# B&R Automation Studio project VisionSample (part 5)

#### Main.st
```iecst
// --------------------------------------------------------------------------------------------------------------------
// General vision task. This is a support task for the mappVision. The following functions are implemneted
// - Translate some values in text messages
// - Reset camera trigger when inspection is finsihed
// - Load vision application
// - Save diagnostic data
// Version 2.x (Check revision history for details)
// --------------------------------------------------------------------------------------------------------------------
PROGRAM _INIT

	userInitCommonPreAction;

	FOR idx:= START_IDX TO MAX_NUM_CAMS BY 1 DO
		setupPointersAction;

		//  Create IO path to cam
		this.path := 'IF3.ST';
		tmpStr := USINT_TO_STRING(idx);
		brsstrcat(ADR(this.path),ADR(tmpStr));

		this.recipePVName := '::Vision1:hmiInstance[';
		brsstrcat(ADR(this.recipePVName),ADR(tmpStr));
		brsstrcat(ADR(this.recipePVName),ADR('].in.recipe'));

		// Create IO path to lights
		FOR i := START_IDX TO MAX_NUM_LIGHTS BY 1 DO
			this.lightPath[i] := 'IF3.ST';
			tmpStr := USINT_TO_STRING(idx*16+(i-1));
			brsstrcat(ADR(this.lightPath[i]),ADR(tmpStr));
		END_FOR

		FOR i:= START_IDX TO MAX_NUM_RESULTS BY 1 DO
			hmi.out.tableVF.tableNum[i] := i;
		END_FOR

		hmi.out.wsPort := 18000+idx*10;
		this.mappView.enable := TRUE;
		this.mappView.wsPort := hmi.out.wsPort;
		this.mappView.simulateConfig.activate := DiagCpuIsSimulated();
		this.mappView.simulateConfig.pFile := ADR('img');
		this.mappView.simulateConfig.useRandomNumbers := FALSE;
		this.mappView.simulateConfig.appendNumber := TRUE;
		this.mappView.simulateConfig.autoIncrementNumber := TRUE;
		this.mappView.simulateConfig.minNumber := 1;
		this.mappView.simulateConfig.maxNumber := 3;

		this.visionDiagFileDevice := 'VI_DIAG'; // File device is created in Files program (changes to USB if such is pluged in)

		hmi.out.camera.plNodeNr := idx;
		hmi.in.recipe.cam.focus := 200;
		hmi.in.recipe.cam.exposureTime := 100;

		hmi.in.cmd.resetInfo := TRUE;

		// -----------------------------------------------------------------------------------------------------------
		// Set camera specific data
		// -----------------------------------------------------------------------------------------------------------

		hmi.in.cmd.resultTabIndex := 5;
		CASE idx OF
			1:
				this.mappView.pMappLink := ADR(gCameraBlob);
				this.mappView.simulateConfig.pDevice := ADR('SIM_BLOB');
				hmi.out.camera.visionFunction := 'BLOB';
				hmi.out.usedVF.BLOB := TRUE;
				hmi.in.cmd.resultTabIndex := MIN(hmi.in.cmd.resultTabIndex,idx-1);
			2:
				this.mappView.pMappLink := ADR(gCameraCodeReading);
				this.mappView.simulateConfig.pDevice := ADR('SIM_CR');
				hmi.out.camera.visionFunction := 'Code Reader';
				hmi.out.usedVF.codeReader := TRUE;
				hmi.in.cmd.resultTabIndex := MIN(hmi.in.cmd.resultTabIndex,idx-1);
				(*hmi.out.VF.numResults*)
			3:
				this.mappView.pMappLink := ADR(gCameraMatch);
				this.mappView.simulateConfig.pDevice := ADR('SIM_MATCH');
				hmi.out.camera.visionFunction := 'Matching';
				hmi.out.usedVF.matching := TRUE;
				hmi.in.cmd.resultTabIndex := MIN(hmi.in.cmd.resultTabIndex,idx-1);
			4:
				this.mappView.pMappLink := ADR(gCameraMeasurement);
				this.mappView.simulateConfig.pDevice := ADR('SIM_MEAS');
				hmi.out.camera.visionFunction := 'Measurement';
				hmi.out.usedVF.measurement := TRUE;
				hmi.in.cmd.resultTabIndex := MIN(hmi.in.cmd.resultTabIndex,idx-1);
			5:
				this.mappView.pMappLink := ADR(gCameraOCR);
				this.mappView.simulateConfig.pDevice := ADR('SIM_OCR');
				hmi.out.camera.visionFunction := 'OCR';
				hmi.out.usedVF.OCR := TRUE;
				hmi.in.cmd.resultTabIndex := MIN(hmi.in.cmd.resultTabIndex,idx-1);
			6:
				this.mappView.pMappLink := ADR(gCameraPxl);
				this.mappView.simulateConfig.pDevice := ADR('SIM_PXCNT');
				hmi.out.camera.visionFunction := 'Pixel Counter';
				hmi.out.usedVF.pixelCounter := TRUE;
				hmi.in.cmd.resultTabIndex := MIN(hmi.in.cmd.resultTabIndex,idx-1);

		END_CASE

		userInitLocalPostAction;

	END_FOR

END_PROGRAM

// -----------------------------------------------------------------------------------------------------------
// Cyclic part
// -----------------------------------------------------------------------------------------------------------
PROGRAM _CYCLIC

	userCommonPreAction; // user common action before all other

	FOR idx:= START_IDX TO MAX_NUM_CAMS BY 1 DO
		setupPointersAction;

		userLocalPreAction; // user local action before all other

		// -----------------------------------------------------------------------------------------------------------
		// Translate camera status in readable text
		// -----------------------------------------------------------------------------------------------------------
		IF hw.camera.in.common.moduleOk THEN
			brdkViBase_camStatusToString(hw.camera.in.status.cameraStatus,ADR(hmi.out.camera.statusText));
		ELSE
			hmi.out.camera.statusText := 'Disconnected';
		END_IF

		// -----------------------------------------------------------------------------------------------------------
		// Check if vision cockpit is open
		// -----------------------------------------------------------------------------------------------------------
		hmi.out.camera.mappVisionActive := (hw.camera.in.status.cameraStatus AND 16#8000_0000) > 0;

		// -----------------------------------------------------------------------------------------------------------
		// Read camera hardware info
		// -----------------------------------------------------------------------------------------------------------

		IF hmi.in.cmd.resetInfo THEN
			hmi.in.cmd.resetInfo := FALSE;
			hmi.in.cameraInfo.distance := hmi.in.recipe.cam.focus;
			this.brdkViBase_getCameraInfo_0.execute := TRUE;
			this.brdkViBase_getCameraInfo_0.pluggedModule := hw.camera.in.common.moduleOk AND NOT DiagCpuIsSimulated();

			FOR i := START_IDX TO MAX_NUM_LIGHTS BY 1 DO
				this.brdkViBase_getLightInfo[i].execute := TRUE;
				this.brdkViBase_getLightInfo[i].pInfo := ADR(hmi.out.lights[i].info);
				this.brdkViBase_getLightInfo[i].pDevicePath := ADR(this.lightPath[i]);
				this.brdkViBase_getLightInfo[i].pluggedModule := hw.lights[i].in.common.moduleOk AND NOT DiagCpuIsSimulated();
			END_FOR

		END_IF

		this.brdkViBase_getCameraInfo_0.pDevicePath := ADR(this.path);
		this.brdkViBase_getCameraInfo_0.pInfo := ADR(hmi.in.cameraInfo);
		this.brdkViBase_getCameraInfo_0();

		FOR i:=START_IDX TO MAX_NUM_LIGHTS BY 1 DO
			this.brdkViBase_getLightInfo[i]();

			IF hmi.out.lights[i].info.orderNr <> '' AND this.brdkViBase_getLightInfo[i].status = ERR_OK THEN
				// set Camera flash options based on current camera
				brdkViBase_LEDColorToOptions(hmi.out.lights[i].info.LED_color, ADR(hmi.out.lights[i].flashLightOptions));
			END_IF
		END_FOR

		IF hw.camera.out.par.focus <> hmi.in.recipe.cam.focus THEN
			hmi.in.cameraInfo.distance := hmi.in.recipe.cam.focus;
		END_IF

		IF hmi.in.cameraInfo.orderNr <> '' AND this.brdkViBase_getCameraInfo_0.status = ERR_OK THEN
			brdkViBase_calcOpticInfo(hmi.in.cameraInfo, hmi.out.camera.opticInfo); // calculate optic info based on defined info

			// set Camera flash options based on current camera
			brdkViBase_LEDColorToOptions(hmi.in.cameraInfo.LED_color, ADR(hmi.out.camera.flashLightOptions));
		END_IF

		IF hw.io.in.nettime > this.axisTrig.nettimeLastCycle_us THEN
			this.axisTrig.powerlinkCycle_us	:= hw.io.in.nettime - this.axisTrig.nettimeLastCycle_us;
		ELSE
			this.axisTrig.powerlinkCycle_us	:= -2147483648-hw.io.in.nettime + 2147483647-this.axisTrig.nettimeLastCycle_us; // handle wrap around
		END_IF
		this.axisTrig.nettimeLastCycle_us	:= hw.io.in.nettime;

		// -----------------------------------------------------------------------------------------------------------
		// Image trigger (camera and lights)
		// -----------------------------------------------------------------------------------------------------------
		hmi.in.recipe.cam.flashColor := STRING_TO_USINT(hmi.in.recipe.cam.flashColorStr);
		hw.camera.out.par.focus 			:= hmi.in.recipe.cam.focus;
		hw.camera.out.par.flashSegment	 	:= hmi.in.recipe.cam.flashSegment;
		hw.camera.out.par.flashColor 		:= hmi.in.recipe.cam.flashColor;
		hw.camera.out.par.exposureTime 		:= hmi.in.recipe.cam.exposureTime;
		hw.camera.out.par.chromaticLock 	:= hmi.in.recipe.cam.chromaticLock;
		hw.camera.out.par.gainLevel 		:= hmi.in.recipe.cam.gainLevel;
		hw.camera.out.par.IRFilter			:= hmi.in.recipe.cam.IRFilter;

		//-------------------------------------------------------------------------

		// Copy recipe data (e.g. enable, maximal number of results, etc.)
		hw.VF.blob.out			:=hmi.in.recipe.BLOB;
		hw.VF.codeReader.out	:= hmi.in.recipe.CR;
		hw.VF.matching.out		:=hmi.in.recipe.match;
		hw.VF.measurement.out	:=hmi.in.recipe.meassurement;
		hw.VF.ocr.out			:=hmi.in.recipe.OCR;
		hw.VF.pixelCnt.out		:=hmi.in.recipe.pxCnt;

		hmi.out.camera.processingTime:=hw.camera.in.status.cameraProcessingTime;

		CASE idx OF
			1:
				hmi.out.VF.processingTime := hw.VF.blob.in.common.functionProcessingTime;
				hmi.out.VF.numResults := hw.VF.blob.in.common.numResults;
			2:
				hmi.out.VF.processingTime := hw.VF.codeReader.in.common.functionProcessingTime;
				hmi.out.VF.numResults := hw.VF.codeReader.in.common.numResults;
			3:
				hmi.out.VF.processingTime := hw.VF.matching.in.common.functionProcessingTime;
				hmi.out.VF.numResults := hw.VF.matching.in.common.numResults;
			4:
				hmi.out.VF.processingTime := hw.VF.measurement.in.common.functionProcessingTime;
				hmi.out.VF.numResults := hw.VF.measurement.in.common.numResults;
			5:
				hmi.out.VF.processingTime := hw.VF.ocr.in.common.functionProcessingTime;
				hmi.out.VF.numResults := hw.VF.ocr.in.common.numResults;
			6:
				hmi.out.VF.processingTime := hw.VF.pixelCnt.in.common.functionProcessingTime;
				hmi.out.VF.numResults := hw.VF.pixelCnt.in.common.numResults;
		END_CASE;

		//-------------------------------------------------------------------------

		this.ioTrigger(CLK := hw.io.in.commonTrigger OR NOT hw.io.in.individualTrigger);
		this.repetitiveTriggerTON.IN := hmi.in.recipe.repetitiveTrigger;
		this.repetitiveTriggerTON.PT := UDINT_TO_TIME(hmi.in.recipe.repetitiveTriggerInterval);
		this.repetitiveTriggerTON();

		// check if camera is ready for an image trigger and MappView have been updated
		IF this.brdkViBase_imgTrigger_0.ready AND NOT this.brdkViBase_imgTrigger_0.busy AND this.mappView.status = 0 THEN

			// Hmi manual trigger
			IF hmi.in.cmd.trigger OR this.repetitiveTriggerTON.Q THEN
				hmi.in.cmd.trigger 							:= FALSE;

				this.repetitiveTriggerTON(IN:=FALSE);

				this.brdkViBase_imgTrigger_0.trigger 		:= TRUE;
				this.brdkViBase_imgTrigger_0.delayNettime 	:= hw.io.in.nettime + gAxis.status.powerlinkCycleTime * 12+10000; // Calc nettime close to currnet time
				this.currentTriggerNum := 1;
				// Axis trigger
			ELSIF hmi.in.recipe.enableAxisTrigger AND
				gAxis.status.triggerTimeDelta >= (commonHmi.in.recipe.visionPreTriggerCycles * this.axisTrig.powerlinkCycle_us) AND
				gAxis.status.triggerTimeDelta <= ((commonHmi.in.recipe.visionPreTriggerCycles + 1) * this.axisTrig.powerlinkCycle_us) THEN

				this.brdkViBase_imgTrigger_0.trigger := TRUE;
				this.brdkViBase_imgTrigger_0.delayNettime := gAxis.status.nettime + gAxis.status.triggerTimeDelta; // Use time calculated in Axis program
			ELSIF hmi.in.recipe.enableIoTrigger AND this.ioTrigger.Q THEN

				this.brdkViBase_imgTrigger_0.trigger := TRUE;
				this.brdkViBase_imgTrigger_0.delayNettime :=  hw.io.in.nettime + hmi.in.recipe.ioTriggerDelay ; // Use time calculated in Axis program

			ELSIF this.currentTriggerNum < hmi.in.recipe.multiCaptureNum AND NOT hmi.in.recipe.repetitiveTrigger THEN

				this.brdkViBase_imgTrigger_0.trigger 		:= TRUE;
				this.brdkViBase_imgTrigger_0.delayNettime 	:= hw.io.in.nettime + gAxis.status.powerlinkCycleTime * 12+10000; // Calc nettime close to currnet time

				this.currentTriggerNum := 		this.currentTriggerNum +1;

			END_IF
		END_IF

		this.brdkViBase_imgTrigger_0.searchAcquisitonSettings := hmi.in.cmd.autoSearch;
		this.brdkViBase_imgTrigger_0.pCameraHw := ADR(hw.camera);
		this.brdkViBase_imgTrigger_0.numLights := MAX_NUM_LIGHTS;
		this.brdkViBase_imgTrigger_0.pLightHw := ADR(hw.lights);
		this.brdkViBase_imgTrigger_0.useCamColorForLight := hmi.in.recipe.useCamLedColorForLight;
		this.brdkViBase_imgTrigger_0.useCamExpTimeForLight := hmi.in.recipe.useCamExpTimeForLight;
		this.brdkViBase_imgTrigger_0.simulate.enable := DiagCpuIsSimulated();
		this.brdkViBase_imgTrigger_0.simulate.alwaysSimulateNonePresentLights := TRUE;
		this.brdkViBase_imgTrigger_0.simulate.imgProcessingDelay := T#300ms;
		this.brdkViBase_imgTrigger_0();

		FOR i:=START_IDX TO MAX_NUM_LIGHTS BY 1 DO

			// Manual Light trigger
			// exposuretime
			IF hmi.in.recipe.useCamExpTimeForLight THEN
				hw.lights[i].out.par.exposureTime := hmi.in.recipe.cam.exposureTime;
			ELSE
				hw.lights[i].out.par.exposureTime := hmi.in.recipe.lights[i].exposureTime;
			END_IF
			// color
			IF hmi.in.recipe.useCamLedColorForLight THEN
				hw.lights[i].out.par.flashColor := hmi.in.recipe.cam.flashColor;
			ELSE
				hw.lights[i].out.par.flashColor := hmi.in.recipe.lights[i].flashColor;
			END_IF

			hmi.out.lights[i].common:=hw.lights[i].in.common;
			hmi.out.lights[i].status:=hw.lights[i].in.status;
			hw.lights[i].out.par.flashAngle:=hmi.in.recipe.lights[i].flashAngle;

			hmi.out.lights[i].plNodeNr := idx*16+UINT_TO_USINT(i-1);

			IF hmi.in.cmd.lights[i].flashTrigger AND NOT hw.lights[i].out.cmd.flashTrigger THEN
				hmi.in.cmd.lights[i].flashTrigger := FALSE;
				hw.lights[i].out.cmd.flashTrigger := TRUE;

				// Nettime
				hw.lights[i].out.par.nettime := hw.io.in.nettime + gAxis.status.powerlinkCycleTime * commonHmi.in.recipe.visionPreTriggerCycles;
			ELSIF 	hw.lights[i].out.cmd.flashTrigger AND hw.lights[i].out.par.nettime <= hw.io.in.nettime THEN
				hw.lights[i].out.cmd.flashTrigger := FALSE;
			END_IF
		END_FOR

		// -----------------------------------------------------------------------------------------------------------
		// New image ready and results
		// -----------------------------------------------------------------------------------------------------------
		// New image (hight for one scan)
		IF this.brdkViBase_imgTrigger_0.newImage THEN

			this.mappView.updateImage := NOT hmi.in.recipe.showOnlyLastImage OR this.currentTriggerNum = hmi.in.recipe.multiCaptureNum; // Trigger an update of the image on hmi
			this.DTGetTime_0(enable := TRUE);

			processResultsAction; // Process results action

			userResultProcessingAction; // User defined process results

		END_IF

		// -----------------------------------------------------------------------------------------------------------
		// Selection of specific result
		// -----------------------------------------------------------------------------------------------------------
		IF hmi.in.cmd.click THEN
			hmi.in.cmd.click := FALSE;

			//VF
			brdkStrSubStr(ADR(tmpVF),ADR(hmi.in.cmd.elemId),1,1);
			//ID
			brsstrcpy(ADR(tmpID),ADR(hmi.in.cmd.elemId)+2);

			hmi.in.cmd.intElemId := STRING_TO_USINT(tmpID);
			IF hmi.in.cmd.intElemId > MAX_NUM_RESULTS THEN
				hmi.in.cmd.intElemId := 0;
			END_IF

		END_IF

		IF hmi.in.cmd.intElemId <> this.oldIntElemID THEN
			this.oldIntElemID := hmi.in.cmd.intElemId;
			processResultsAction;
		END_IF

		// -----------------------------------------------------------------------------------------------------------
		// Auto search vision acquistion settings done (save found settings in recipe structure)
		// -----------------------------------------------------------------------------------------------------------

		// search Auto Focus done (hight for one scan)
		IF this.brdkViBase_imgTrigger_0.searchAcquisitonSettingsDone THEN
			hmi.in.cmd.autoSearch 			:= FALSE;
			hmi.in.recipe.cam.gainLevel 	:=	 hw.camera.in.status.gainLevel;
			hmi.in.recipe.cam.focus		 	:=	 hw.camera.in.status.focus;
			hmi.in.recipe.cam.exposureTime 	:=	 hw.camera.in.status.exposureTime;
			this.brdkViBase_imgTrigger_0.searchAcquisitonSettings := FALSE;
			hmi.in.cmd.trigger 				:= TRUE;
		END_IF

		// -----------------------------------------------------------------------------------------------------------
		// MappView get image to show om hmi
		// -----------------------------------------------------------------------------------------------------------

		IF DiagCpuIsSimulated() THEN
			this.mappView.imageFormat := BRDKVIIMG_IMG_TYPE_JPEG;
		ELSE
			this.mappView.imageFormat := commonHmi.in.recipe.imageFormat;
		END_IF
		this.mappView.jpegQuality := commonHmi.in.recipe.jpegQuality;
		this.mappView();

		// -----------------------------------------------------------------------------------------------------------
		// Save image to file devive F:/images
		// -----------------------------------------------------------------------------------------------------------
		CASE this.saveState OF
			0:

				IF (hmi.in.cmd.saveImage OR (this.mappView.newSvgReady AND commonHmi.in.recipe.saveAllImages))  AND gFiles.output.ready THEN
					hmi.in.cmd.saveImage := FALSE;

					// create filename with VF name and current date of the image
					brsstrcpy(ADR(this.tmpFileName),ADR(hmi.out.camera.visionFunction));
					brsstrcat(ADR(this.tmpFileName),ADR('-'));
					brdkViBase_dateTimeToString(this.DTGetTime_0.DT1,'%Y-%m-%d-%H-%M-%S',ADR(this.tmpFileName));

					brsstrcpy(ADR(this.brdkFileWrite.fileName),ADR(this.tmpFileName));

					CASE this.mappView.imageFormat OF
						BRDKVIIMG_IMG_TYPE_JPEG:
							brsstrcat(ADR(this.brdkFileWrite.fileName),ADR('.jpg'));
						BRDKVIIMG_IMG_TYPE_BMP:
							brsstrcat(ADR(this.brdkFileWrite.fileName),ADR('.bmp'));
					END_CASE

					this.brdkFileWrite.enable := TRUE;
					this.brdkFileWrite.dataLength := this.mappView.internal.getImage.destLen;
					this.brdkFileWrite.pData := this.mappView.internal.getImage.pDest;
					this.brdkFileWrite.overwrite := TRUE;
					this.brdkFileWrite.fileDevice := 'IMG';

					this.saveState := 10;
				END_IF
			10:

				IF this.brdkFileWrite.done THEN
					gFiles.input.refresh := TRUE;
					this.brdkFileWrite.enable := FALSE;
					this.saveState := 20;
				END_IF

			20:
				brsstrcpy(ADR(this.brdkFileWrite.fileName),ADR(this.tmpFileName));

				brsstrcat(ADR(this.brdkFileWrite.fileName),ADR('.svg'));
				this.brdkFileWrite.enable := TRUE;
				this.brdkFileWrite.dataLength := brsstrlen(ADR(hmi.out.svgOverlay));
				this.brdkFileWrite.pData := ADR(hmi.out.svgOverlay);
				this.brdkFileWrite.overwrite := TRUE;
				this.brdkFileWrite.fileDevice := 'IMG';

				this.saveState := 30;

			30:
				IF this.brdkFileWrite.done THEN
					gFiles.input.refresh := TRUE;
					this.brdkFileWrite.enable := FALSE;
					this.saveState := 0;
				END_IF

		END_CASE

		this.brdkFileWrite();

		// -----------------------------------------------------------------------------------------------------------
		// Save diagnostic data
		// -----------------------------------------------------------------------------------------------------------
		IF hmi.in.cmd.saveDiagnositc AND gFiles.output.ready THEN
			hmi.in.cmd.saveDiagnositc 			:= FALSE;

			// Delete old file first
			this.fileDelete.enable 					:= TRUE;
			this.fileDelete.pDevice 				:= ADR(this.visionDiagFileDevice);
			this.fileDelete.pName 					:= ADR(hmi.in.diagnosticFilename);

			// Upload diagnostic information
			this.viBaseSaveDiagData_0.MpLink 		:= this.mappView.pMappLink;
			this.viBaseSaveDiagData_0.DeviceName 	:= ADR(this.visionDiagFileDevice);
			this.viBaseSaveDiagData_0.FileName 		:= ADR(hmi.in.diagnosticFilename);
			hmi.out.camera.saveDiagStatus 			:= UINT_TO_DINT(ERR_FUB_BUSY);
		END_IF

		// file delete done or error (if file do not exsist)
		IF (this.fileDelete.enable AND this.fileDelete.status = ERR_OK) THEN
			this.fileDelete.enable 				:= FALSE;
			this.viBaseSaveDiagData_0.Execute 	:= TRUE;
		END_IF

		// Done
		IF (this.viBaseSaveDiagData_0.Done) THEN
			hmi.out.camera.saveDiagStatus		:= UINT_TO_DINT(ERR_OK);
			this.viBaseSaveDiagData_0.Execute 	:= FALSE;
		END_IF

		// Error
		IF (NOT this.viBaseSaveDiagData_0.Busy AND this.viBaseSaveDiagData_0.Error) THEN
			hmi.out.camera.saveDiagStatus		:= this.viBaseSaveDiagData_0.StatusID;
			this.viBaseSaveDiagData_0.Execute 	:= FALSE;
		END_IF

		this.viBaseSaveDiagData_0();
		this.fileDelete();

		// -----------------------------------------------------------------------------------------------------------
		// Get Vision application list from camera
		// -----------------------------------------------------------------------------------------------------------

		// trigger
		IF hmi.in.cmd.vaList.refresh THEN
			hmi.in.cmd.vaList.refresh 	:= FALSE;

			this.getVaList.Execute 		:= TRUE;
			this.getVaList.Format 		:= viBASE_FORMAT_PLAIN_TEXT;
			this.getVaList.List 		:= ADR(hmi.out.vaList.list);
			this.getVaList.ListLen 		:= SIZEOF(hmi.out.vaList.list);
			this.getVaList.MpLink 		:= this.mappView.pMappLink;
		END_IF

		// Done
		IF this.getVaList.Done THEN
			this.getVaList.Execute 		:= FALSE;
			hmi.out.vaList.length 		:= this.getVaList.NrEntries;
		END_IF

		// Error
		IF this.getVaList.Error THEN
			this.getVaList.Execute 		:= FALSE;
			hmi.out.vaList.lastError 	:= this.getVaList.StatusID;
		END_IF

		this.getVaList();

		// -----------------------------------------------------------------------------------------------------------
		// Load vision application
		// -----------------------------------------------------------------------------------------------------------

		// Trigger
		IF hmi.in.cmd.vaList.load AND brsstrlen(ADR(hmi.out.vaList.list[hmi.in.cmd.vaList.selectedIndex])) > 5 THEN
			hmi.in.cmd.vaList.load 						:= FALSE;

			this.viBaseLoadApplication_0.Execute 	:= TRUE;
			this.viBaseLoadApplication_0.MpLink		:= this.mappView.pMappLink;
			this.viBaseLoadApplication_0.Name		:= ADR(hmi.out.vaList.list[hmi.in.cmd.vaList.selectedIndex]);
			hmi.out.camera.vaLoad 					:= UINT_TO_DINT(ERR_FUB_BUSY);
		ELSE
			hmi.in.cmd.vaList.load := FALSE;
		END_IF

		// Done
		IF (this.viBaseLoadApplication_0.Done) THEN
			hmi.in.cmd.vaList.selectedIndex := 0;
			this.viBaseLoadApplication_0.Execute 	:= FALSE;
			hmi.out.camera.vaLoad 					:= UINT_TO_DINT(ERR_OK);
		END_IF

		// Error
		IF (NOT this.viBaseLoadApplication_0.Busy AND this.viBaseLoadApplication_0.Error) THEN
			this.viBaseLoadApplication_0.Execute 	:= FALSE;
			hmi.out.camera.vaLoad 					:= this.viBaseLoadApplication_0.StatusID;
		END_IF

		this.viBaseLoadApplication_0();

		// -----------------------------------------------------------------------------------------------------------
		// HMI stuff
		// -----------------------------------------------------------------------------------------------------------
		hmiAction;

		// -----------------------------------------------------------------------------------------------------------
		// Recipe handling (register recipse data structure
		// -----------------------------------------------------------------------------------------------------------
		this.mpRecipeRegVar.Enable 		:= gRecipe.out.active;
		this.mpRecipeRegVar.MpLink 		:= gRecipe.out.mpLink;
		this.mpRecipeRegVar.ConfirmSave := this.mpRecipeRegVar.SaveNotification;
		this.mpRecipeRegVar.Category 	:= ADR('Recipe');
		this.mpRecipeRegVar.PVName 		:= ADR(this.recipePVName);
		this.mpRecipeRegVar();

		// handle conversion from CR dropDown value to interger and back
		IF this.mpRecipeRegVar.UpdateNotification THEN
			hmi.in.recipe.CRTypeStr := USINT_TO_STRING(hmi.in.recipe.CR.symbolType);

			FOR i:=START_IDX TO MAX_NUM_LIGHTS BY 1 DO
				this.brdkViBase_getLightInfo[i]();
				hmi.in.cmd.lightColorStr[i] := USINT_TO_STRING(hmi.in.recipe.lights[i].flashColor );
			END_FOR

		ELSE
			hmi.in.recipe.CR.symbolType := STRING_TO_USINT(hmi.in.recipe.CRTypeStr);
			FOR i:=START_IDX TO MAX_NUM_LIGHTS BY 1 DO
				this.brdkViBase_getLightInfo[i]();
				hmi.in.recipe.lights[i].flashColor := STRING_TO_USINT(hmi.in.cmd.lightColorStr[i]);
			END_FOR
		END_IF

		// Clear ready for init (auto load) if data structures have not been registred
		IF NOT this.mpRecipeRegVar.Active THEN
			gRecipe.in.readyForInit := FALSE;
		END_IF

		userLocalPostAction; // user local action after all other

	END_FOR

	userCommonPostAction; // user common action after all other

	// -----------------------------------------------------------------------------------------------------------
	//Configure the pointers (this,hmi,hw etc.) show the correct data for that watch index
	// -----------------------------------------------------------------------------------------------------------
	watchIdx := LIMIT(START_IDX,watchIdx,MAX_NUM_CAMS);
	idx := watchIdx;
	setupPointersAction;

					END_PROGRAM

PROGRAM _EXIT

	FOR idx:= START_IDX TO MAX_NUM_CAMS BY 1 DO
		setupPointersAction;

		this.mappView(enable := FALSE);
		this.mpRecipeRegVar(Enable := FALSE);

		userExitLocalPostAction;
	END_FOR

	userExitCommonPostAction;

					END_PROGRAM
```

### VisionTypes.typ
```iecst
(*-----------------------------------------------------------------------------------------------------------------------------------------*)
(*General vision structures*)

TYPE
	typVisionMain : 	STRUCT
		CMD : typVisionCommand;
		CFG : typVisionConfig;
		DAT : typVisionData;
		HW : typVisionHW;
	END_STRUCT;
	typVisionCommand : 	STRUCT
		ImageTrigger : BOOL;
		ImageTriggerReset : BOOL;
		AutoSetupStartStop : BOOL;
	END_STRUCT;
	typVisionConfig : 	STRUCT
		VisionFunction : enumVisionFunction;
		PowerlinkNode : USINT;
		DataStructure : UDINT;
		ComponentLink : ViComponentType;
		ResolutionWidth : UINT; (*Nr of sensor pixels in x direction (width). Is always bigger than height*)
		ResolutionHeight : UINT; (*Nr of sensor pixels in y direction (height). Is always smaller than width*)
	END_STRUCT;
	typVisionData : 	STRUCT
		Enable : BOOL := FALSE;
		MaxItemCnt : USINT := 10;
		NettimeDelay : DINT;
		Timeout : UINT := 5000;
		Gain : USINT;
		Focus : UINT;
		Exposure : UDINT;
		FlashColor : USINT := 1;
		FlashSegment : USINT := 15;
		LedColor : USINT;
		IRFilter : BOOL;
		OffsetROIX : DINT;
		OffsetROIY : DINT;
		OffsetROIRotationCenterX : DINT;
		OffsetROIRotationCenterY : DINT;
		OffsetROIOrientation : INT;
		ChromaticLock : BOOL;
		Alignment : USINT;
		AutoSetupGain : USINT;
		AutoSetupFocus : UINT;
		AutoSetupExposure : UDINT;
		AcquisitionAcceptedCnt : USINT;
		AcquisitionCompletedCnt : USINT;
		AcquisitionFailedCnt : USINT;
		LightWarningCnt : USINT;
		ImageProcessingError : UINT;
		ImageProcessingActive : BOOL;
		ImageNettime : DINT;
		ProcessingTimeCamera : UINT;
		ProcessingTimeFunction : UINT;
		ResultCnt : USINT;
		CockpitIsActive : BOOL;
		Status : UDINT;
		StatusText : STRING[30];
		Active : BOOL;
	END_STRUCT;
	typVisionHW : 	STRUCT
		Connected : BOOL;
		Ready : BOOL;
		DigitalInput01 : BOOL;
		DigitalOutput01 : BOOL;
		DigitalOutputStatus01 : BOOL;
		DigitalOutput02 : BOOL;
		DigitalOutputStatus02 : BOOL;
		SerialNumber : UDINT;
		ID : UDINT;
		Variant : UDINT;
		Firmware : UDINT;
		Undervoltage : BOOL;
		Temperature : SINT;
	END_STRUCT;
	enumVisionFunction :
		(
		enumFunctionNone,
		enumBlob,
		enumCoderReader,
		enumMatch,
		enumMeasurement,
		enumOCR,
		enumDOCR,
		enumPixelCounter
		);
END_TYPE

(*-----------------------------------------------------------------------------------------------------------------------------------------*)
(*General Light structures*)

TYPE
	typLightMain : 	STRUCT
		CMD : typLightCommand;
		CFG : typLightConfig;
		DAT : typLightData;
		HW : typLightHW;
	END_STRUCT;
	typLightCommand : 	STRUCT
		FlashTrigger : BOOL;
		FlashTriggerReset : BOOL;
	END_STRUCT;
	typLightConfig : 	STRUCT
		LightType : enumLightType;
		PowerlinkNode : USINT;
	END_STRUCT;
	typLightData : 	STRUCT
		Enable : USINT := 1;
		FlashColor : USINT := 1;
		FlashSegment : UINT := 15;
		Exposure : UDINT := 200;
		SetAngle : UINT;
		Timeout : UINT := 5000;
		NettimeDelay : DINT;
		FlashAcceptedCnt : USINT;
		FlashCompletedCnt : USINT;
		FlashFailedCnt : USINT;
		Status : UDINT;
	END_STRUCT;
	typLightHW : 	STRUCT
		Connected : BOOL;
		Ready : BOOL;
		SerialNumber : UDINT;
		ID : UDINT;
		Variant : UDINT;
		Firmware : UDINT;
		TemperatureLED : SINT;
		TemperatureControllerBoard : SINT;
		WarningCnt : USINT;
	END_STRUCT;
	enumLightType :
		(
		enumLightNone,
		enumBacklight,
		enumLightbar
		);
END_TYPE

(*-----------------------------------------------------------------------------------------------------------------------------------------*)
(*General nettime structures*)

TYPE
	typVisionNettime : 	STRUCT
		CMD : typNettimeCommand;
		CFG : typNettimeConfig;
		DAT : typNettimeData;
	END_STRUCT;
	typNettimeCommand : 	STRUCT
		Activate : BOOL;
	END_STRUCT;
	typNettimeConfig : 	STRUCT
		AxisPeriod : LREAL; (*Units when period repeats*)
		AxisPositionTrigger : LREAL; (*Position in the period where trigger is fired*)
		AxisPositionDelay_Cycles : LREAL; (*Delay in PLK cycles for the read position from drive*)
		VisionPreTrigger_Cycles : DINT; (*Number of powerlink cycles the trigger has to be send ahead*)
	END_STRUCT;
	typNettimeData : 	STRUCT
		NettimeNext_us : DINT; (*Calculated nettime for next trigger*)
		NettimeDelta_us : DINT; (*Difference between current nettime and calculated nettime for the camera trigger*)
		AxisPosition : LREAL; (*Current axis position*)
		AxisVelocity : LREAL; (*Current axis position*)
		AxisInVelocity : BOOL; (*Indicates that the axis is moving at speed*)
		Overflow : DINT; (*Counts up when a trigger could not be set on time*)
	END_STRUCT;
END_TYPE

(*-----------------------------------------------------------------------------------------------------------------------------------------*)
(*Image upload structures*)

TYPE
	typVisionImage : 	STRUCT
		CMD : typVisionImageCommand;
		CFG : typVisionImageConfig;
		DAT : typVisionImageData;
	END_STRUCT;
	typVisionImageCommand : 	STRUCT
		CreateDir : BOOL;
		DeleteDir : BOOL;
		DeleteImage : BOOL;
		GetImage : BOOL;
		SaveImage : BOOL;
		Refresh : BOOL;
		ResetError : BOOL;
	END_STRUCT;
	typVisionImageConfig : 	STRUCT
		FileDevice : STRING[80];
		FileName : STRING[80];
		DirName : STRING[80];
		ImageQuality : USINT := 50;
		ImageHeight : UINT := 1280;
		ImageWidth : UINT := 1024;
		ImageType : ViBaseImageTypeEnum;
		ComponentLink : ViComponentType;
	END_STRUCT;
	typVisionImageData : 	STRUCT
		ImagesList : ARRAY[0..19]OF STRING[80];
		ImageSelected : STRING[80];
		ImagePath : STRING[80];
		Crosshair : ARRAY[1..MAX_NUM_RESULTS]OF typVisionImageDataCrosshair;
		Status : DINT;
	END_STRUCT;
	typVisionImageDataCrosshair : 	STRUCT
		CrosshairX : REAL;
		CrosshairY : REAL;
		CrosshairRotate : REAL;
		Text : STRING[1000];
	END_STRUCT;
END_TYPE

(*-----------------------------------------------------------------------------------------------------------------------------------------*)
(*Vision specific structures*)

TYPE
	typCodeReaderMain : 	STRUCT  (*Code reader structures*)
		CodeType : USINT;
		GradingEnable : BOOL;
		RobustnessEnable : BOOL;
		ParameterMode : USINT;
		ParameterOptimization : USINT;
		BarcodeText : ARRAY[1..MAX_NUM_RESULTS]OF STRING[100];
		BarcodeType : ARRAY[1..MAX_NUM_RESULTS]OF USINT;
		PositionX : ARRAY[1..MAX_NUM_RESULTS]OF DINT;
		PositionY : ARRAY[1..MAX_NUM_RESULTS]OF DINT;
		Orientation : ARRAY[1..MAX_NUM_RESULTS]OF INT;
		Grading : ARRAY[1..MAX_NUM_RESULTS]OF SINT;
		EnhancedGrading : ARRAY[1..23]OF USINT;
	END_STRUCT;
	typBlobMain : 	STRUCT  (*Blob function structures*)
		RegionalFeature : BOOL;
		EnhancedBlobInformation : BOOL := FALSE;
		ModelNumber : ARRAY[1..MAX_NUM_RESULTS]OF USINT;
		Clipped : ARRAY[1..MAX_NUM_RESULTS]OF BOOL;
		Area : ARRAY[1..MAX_NUM_RESULTS]OF UDINT;
		PositionX : ARRAY[1..MAX_NUM_RESULTS]OF DINT;
		PositionY : ARRAY[1..MAX_NUM_RESULTS]OF DINT;
		Orientation : ARRAY[1..MAX_NUM_RESULTS]OF INT;
		MeanGrayValue : ARRAY[1..MAX_NUM_RESULTS]OF USINT;
		Length : ARRAY[1..MAX_NUM_RESULTS]OF UDINT;
		Width : ARRAY[1..MAX_NUM_RESULTS]OF UDINT;
	END_STRUCT;
	typMatchMain : 	STRUCT  (*Match function structures*)
		MinScore : USINT := 70;
		MaxOverlap : USINT;
		ModelNumber : ARRAY[1..MAX_NUM_RESULTS]OF USINT;
		Score : ARRAY[1..MAX_NUM_RESULTS]OF USINT;
		PositionX : ARRAY[1..MAX_NUM_RESULTS]OF DINT;
		PositionY : ARRAY[1..MAX_NUM_RESULTS]OF DINT;
		Orientation : ARRAY[1..MAX_NUM_RESULTS]OF INT;
		Scale : ARRAY[1..MAX_NUM_RESULTS]OF USINT;
		RotCenterX : ARRAY[1..MAX_NUM_RESULTS]OF DINT;
		RotCenterY : ARRAY[1..MAX_NUM_RESULTS]OF DINT;
	END_STRUCT;
	typOCRMain : 	STRUCT  (*OCR function structures*)
		ParameterMode : USINT;
		GradingEnable : BOOL;
		Text : ARRAY[1..MAX_NUM_RESULTS]OF STRING[50];
		Grading : ARRAY[1..MAX_NUM_RESULTS]OF USINT;
		PositionX : ARRAY[1..MAX_NUM_RESULTS]OF DINT;
		PositionY : ARRAY[1..MAX_NUM_RESULTS]OF DINT;
		Orientation : ARRAY[1..MAX_NUM_RESULTS]OF INT;
	END_STRUCT;
	typDOCRMain : 	STRUCT  (*OCR function structures*)
		MinConfidence : USINT := 20;
		Text : ARRAY[1..MAX_NUM_RESULTS]OF STRING[25];
		MinConfidenceROI : ARRAY[1..MAX_NUM_RESULTS]OF USINT;
		NumDiscardedCharacters : ARRAY[1..MAX_NUM_RESULTS]OF USINT;
		PositionX : ARRAY[1..MAX_NUM_RESULTS]OF DINT;
		PositionY : ARRAY[1..MAX_NUM_RESULTS]OF DINT;
		Orientation : ARRAY[1..MAX_NUM_RESULTS]OF INT;
	END_STRUCT;
	typPixelMain : 	STRUCT  (*OCR function structures*)
		EnhancedPixelCounterInformation : BOOL := FALSE;
		ModelNumber : ARRAY[1..MAX_NUM_RESULTS]OF USINT;
		NumPixels : ARRAY[1..MAX_NUM_RESULTS]OF UDINT;
		MinGray : ARRAY[1..MAX_NUM_RESULTS]OF USINT;
		MaxGray : ARRAY[1..MAX_NUM_RESULTS]OF USINT;
		MeanGray : ARRAY[1..MAX_NUM_RESULTS]OF UINT;
		DeviationGray : ARRAY[1..MAX_NUM_RESULTS]OF UINT;
		MedianGray : ARRAY[1..MAX_NUM_RESULTS]OF USINT;
		ModelArea : ARRAY[1..MAX_NUM_RESULTS]OF UDINT;
		NumConnectedComponents : ARRAY[1..MAX_NUM_RESULTS]OF UINT;
		PositionX : ARRAY[1..MAX_NUM_RESULTS]OF DINT;
		PositionY : ARRAY[1..MAX_NUM_RESULTS]OF DINT;
	END_STRUCT;
	typMTMain : 	STRUCT  (*MT function structures*)
		UseResultAsXY : BOOL;
		ParameterMode : USINT;
		Result : ARRAY[1..MAX_NUM_RESULTS]OF DINT;
	END_STRUCT;
END_TYPE
```

### VisionVariables.var
```iecst
(*-----------------------------------------------------------------------------------------------------------------------------------------*)
(*Global variables for sensor hardware and vision functions*)
VAR
	gBlob : typBlobMain; (*Data that is specific for the blob function*)
	gCodeReader : typCodeReaderMain; (*Data that is specific for the code reader*)
	gMatch : typMatchMain; (*Data that is specific for the match function*)
	gMT : typMTMain; (*Data that is specific for the measurement function*)
	gOCR : typOCRMain; (*Data that is specific for the OCR function*)
	gDOCR : typDOCRMain; (*Data that is specific for the OCR function*)
	gPixel : typPixelMain; (*Data that is specific for the Pixel Counter function*)
	gVisionImage : typVisionImage; (*Data for image handling*)
	gVisionLight : ARRAY[0..MAX_NUM_LIGHTS] OF typLightMain; (*General Light  functions that are independent from the inspection function*)
	gVisionNettime : typVisionNettime; (*Data for nettime calculation*)
	gVisionSensor : ARRAY[0..MAX_NUM_CAMS] OF typVisionMain; (*General vision functions that are independent from the inspection function*)
	gSelectedSensor : UINT := 1; (*Selected camera node number*)
	gSelectedLight : UINT := 1; (*Selected Light node number*)
	NettimeCurrent_us : DINT; (*Current Powerlink nettime*)
END_VAR
(*-----------------------------------------------------------------------------------------------------------------------------------------*)
(*Global constants*)
VAR CONSTANT
	MAX_NUM_CAMS : UINT := 7; (*Maximum number of camera's*)
	MAX_NUM_LIGHTS : UINT := 5; (*Maximum number of light's*)
	MAX_NUM_RESULTS : UINT := 10; (*Maximum number of results*)
	MAX_NUM_PRODUCTS : UINT := 8; (*Maximum number of products for color detection*)
	MAX_IDX_VA_LIST : UINT := 19; (*Maximum number of entrys in the Vision Application list*)
	CONVERT_CYCLES : UINT := 2000;
	DEVICE_NAME : STRING[40] := 'VisionFileDevice'; (*File device where the images and recipes are stored*)
	NETTIME_DEFAULT_DELAY : UDINT := 30000; (*This delay is used when software trigger is used and nettime is enabled*)
	NETTIME_ENABLE : BOOL := FALSE; (*Enable nettime code, this generates the nettime when using manual triggers*)
	MAX_NUM_CODETYPES : USINT := 69; (*Maximum number of code types*)
END_VAR
VAR
	CodeTypes : {REDUND_UNREPLICABLE} ARRAY[0..MAX_NUM_CODETYPES] OF STRING[80] := ['Auto Identify (0)','2/5 Industrial (1)','2/5 Interleaved (2)','Codebar (3)','Code 32 (4)','Code 39 (5)','Code 93 (6)','Code 128 (7)','MSI (8)','PharmaCode (9)','EAN-8 (10)','EAN-8 Add-On 2 (11)','EAN-8 Add-On 5 (12)','EAN-13 (13)','EAN-13 Add-On 2 (14)','EAN-13 Add-On 5 (15)',4(''),'UPC-A (20)','UPC-A Add-On 2 (21)','UPC-A Add-On 5 (22)','UPC-E (23)','UPC-E Add-On 2 (24)','UPC-E Add-On 5 (25)',4(''),'GS1-128 (30)','GS1 DataBar Omnidirectional (31)','GS1 DataBar Truncated (32)','GS1 DataBar Stacked (33)','GS1 DataBar Stacked Omnidirectional (34)','GS1 DataBar Limited (35)','GS1 DataBar Expanded (36)','GS1 DataBar ExpandedStacked (37)',12(''),'Data Matrix ECC200 (50)','QR Code Model 1 (51)','QR Code Model 2 (52)','Micro QRCode (53)','PDF417 (54)','Aztec Code (55)',4(''),'GS1 Data Matrix (60)','GS1 QR Code Model 1 (61)','GS1 QR Code Model 2 (62)','GS1 Aztec Code (63)',6('')]; (*Codes types for code reading*)
END_VAR
```

### revision.txt
```
Version 5.28 (15.01.2022)
- Update to mappVision 5.28
- Added Deep OCR sample
- Fixed height and width for crosshairs

Version 5.26.3 (03.07.2024)
- Fixed artefacts in main page image when no camera image was loaded
- Use vision sensor resolution from config to account for cameras with higher resolution

Version 5.26.2 (10.06.2024)
- Optimized image download
- General code optimizations

Version 5.26.1
- Update to mappVision 5.26
- Changed image request to official function block
- Removed recipe management
- Removed color detection
- Removed optic details
- Removed VC4 support
- Removed TCP proxy task
- Removed function to load VA applications
- Removed function to download images
```

### Program Logical/Vision/Axis

#### Main.st
```iecst
// --------------------------------------------------------------------------------------------------------------------
// Motion sample for using nettime
// --------------------------------------------------------------------------------------------------------------------
PROGRAM _INIT
	gAxis_1;
	gAxis_2;

	MpAxisBasic_0.Enable			:= TRUE;
	MpAxisBasic_0.MpLink			:= ADR(gAxis_2);
	MpAxisBasic_0.Parameters		:= ADR(MpAxisBasicPar_0);
	MpAxisBasic_0();
	MpAxisBasicPar_0.Homing.Mode	:= mcHOMING_DEFAULT;
END_PROGRAM

// -----------------------------------------------------------------------------------------------------------
// Cyclic part
// -----------------------------------------------------------------------------------------------------------
PROGRAM _CYCLIC
	MpAxisBasic_0.Power					:= MpAxisBasic_0.Active AND MpAxisBasic_0.Info.ReadyToPowerOn AND cmdAxisPower;
	MpAxisBasic_0.ErrorReset			:= cmdAxisErrorReset;
	MpAxisBasic_0.Home					:= MpAxisBasic_0.PowerOn AND NOT MpAxisBasic_0.IsHomed XOR cmdAxisHome;
	MpAxisBasic_0.MoveVelocity			:= MpAxisBasic_0.PowerOn AND MpAxisBasic_0.IsHomed AND cmdAxisRun;
	IF MpAxisBasic_0.PowerOn AND MpAxisBasic_0.IsHomed AND cmdAxisMoveAbs THEN
		MpAxisBasic_0.MoveAbsolute		:= TRUE;
		MpAxisBasicPar_0.Position		:= gVisionNettime.CFG.AxisPositionTrigger;
	END_IF
	cmdAxisMoveAbs					:= FALSE;
	IF AxisVelocity <> MpAxisBasicPar_0.Velocity OR AxisAcceleration <> MpAxisBasicPar_0.Acceleration THEN
		MpAxisBasicPar_0.Velocity		:= AxisVelocity;
		MpAxisBasicPar_0.Acceleration	:= AxisAcceleration;
		MpAxisBasicPar_0.Deceleration	:= AxisAcceleration;
		MpAxisBasic_0.Update			:= TRUE;
	END_IF
	MpAxisBasic_0();
	gVisionNettime.DAT.AxisInVelocity	:= MpAxisBasic_0.InVelocity;
	gVisionNettime.DAT.AxisPosition		:= MpAxisBasic_0.Position;
	gVisionNettime.DAT.AxisVelocity		:= MpAxisBasic_0.Velocity;
	IF MpAxisBasic_0.UpdateDone THEN
		MpAxisBasic_0.Update := FALSE;
	END_IF
	IF MpAxisBasic_0.InPosition THEN
		MpAxisBasic_0.MoveAbsolute		:= FALSE;
	END_IF
END_PROGRAM
```

### Program Logical/Vision/Vi_image

#### Variables.var
```iecst
VAR CONSTANT
	MAX_ENCODED_SIZE : UDINT := 7000000;
	MAX_IMAGE_SIZE : UDINT := 6500000;
	MAX_CROSSHAIR_SIZE : UDINT := 10000;
END_VAR
VAR
	IMAGE_QUALITY : USINT := 50;
	IMAGE_WIDTH : UINT := 640; (*Image width of the SVG image in mappView*)
	IMAGE_HEIGHT : UINT := 512; (*Image height of the SVG image in mappView*)
END_VAR
(**)
VAR
	Step : VIStep_Enum;
	tmpStr : STRING[80];
	idx : UINT;
END_VAR
(**)
(*File handling*)
VAR
	DirCreate_0 : DirCreate;
	DirDeleteEx_0 : DirDeleteEx;
	FileNamePict : STRING[80];
	FileNameSvg : STRING[80];
	FileCreate_0 : FileCreate;
	FileDelete_0 : FileDelete;
	FileWrite_0 : FileWrite;
	FileClose_0 : FileClose;
	DirRead_0 : DirRead;
	dir_data : fiDIR_READ_DATA;
	dir_entry : UINT;
	file_newest : STRING[80];
	file_oldest : STRING[80];
	date_newest : DATE_AND_TIME;
	date_oldest : DATE_AND_TIME;
	cmdDeleteOldest : BOOL;
	DTGetTime_0 : DTGetTime;
	DTStructure_0 : DTStructure;
	TON_VisPause : TON;
END_VAR
(**)
(*Image handling*)
VAR
	ViBaseGetImage_0 : ViBaseGetImage;
	httpEncodeBase64_0 : httpEncodeBase64;
	bufferImage : ARRAY[0..MAX_IMAGE_SIZE] OF USINT;
	bufferAdr : UDINT;
	bufferLen : UDINT;
	bufferImage64 : ARRAY[0..MAX_IMAGE_SIZE] OF USINT;
	bufferCrosshair : ARRAY[0..MAX_CROSSHAIR_SIZE] OF USINT;
	visImageSelectedOld : STRING[80];
	visCameraImage : STRING[MAX_ENCODED_SIZE];
END_VAR
(**)
```

#### Main.st
```iecst
// --------------------------------------------------------------------------------------------------------------------
// Vision image upload task. This task stores the camera image on the file device media
// Version 2.0
// --------------------------------------------------------------------------------------------------------------------
PROGRAM _INIT
	gVisionImage.CFG.FileDevice 	:= 'VisionFileDevice';		// File device name where the images are stored
	gVisionImage.CFG.DirName		:= 'Vision';				// Directory used for images

	gVisionImage.CMD.CreateDir	:= TRUE;
	gVisionImage.DAT.ImageSelected	:= '';

	brsmemset(ADR(bufferImage), 0, SIZEOF(bufferImage));
	brsmemset(ADR(visCameraImage), 0, SIZEOF(visCameraImage));

END_PROGRAM

// -----------------------------------------------------------------------------------------------------------
// Cyclic part
// -----------------------------------------------------------------------------------------------------------
PROGRAM _CYCLIC

	// -----------------------------------------------------------------------------------------------------------
	// State machine for uploading the image
	// -----------------------------------------------------------------------------------------------------------
	CASE Step OF
		// -----------------------------------------------------------------------------------------------------------
		// Wait for new upload command
		VISTEP_WAIT:
			gVisionImage.DAT.Status := 0;

			// -----------------------------------------------------------------------------------------------------------
			// Create the internal directory VisionImageArchive
			IF gVisionImage.CMD.CreateDir THEN
				gVisionImage.DAT.Status := 65535;
				Step := VISTEP_CREATE_DIR;

				// -----------------------------------------------------------------------------------------------------------
				// Delete image directory
			ELSIF gVisionImage.CMD.DeleteDir THEN
				gVisionImage.DAT.Status := 65535;
				Step := VISTEP_DELETE_DIR;

				// -----------------------------------------------------------------------------------------------------------
			// Refresh image data from file device
			ELSIF gVisionImage.CMD.Refresh THEN
				gVisionImage.DAT.Status := 65535;
				Step := VISTEP_READ_DIR1;

			// -----------------------------------------------------------------------------------------------------------
			// Delete image data from file device
			ELSIF gVisionImage.CMD.DeleteImage THEN
				IF brsstrlen(ADR(gVisionImage.DAT.ImageSelected)) > 0 THEN
					brsstrcpy(ADR(FileNamePict), ADR(gVisionImage.CFG.DirName));
					brsstrcat(ADR(FileNamePict), ADR('/'));
					brsstrcat(ADR(FileNamePict), ADR(gVisionImage.DAT.ImageSelected));
					gVisionImage.DAT.Status := 65535;

					FileDelete_0.enable := FALSE;
					FileDelete_0();

					Step := VISTEP_DELETE_IMAGE;
				ELSE
					gVisionImage.CMD.DeleteImage := FALSE;
				END_IF

				// -----------------------------------------------------------------------------------------------------------
				// Save image from camera
			ELSIF gVisionImage.CMD.GetImage THEN
				ViBaseGetImage_0.Execute := FALSE;
				ViBaseGetImage_0();
				httpEncodeBase64_0.enable := FALSE;
				httpEncodeBase64_0();

				gVisionImage.DAT.Status		:= 65535;
				Step						:= VISTEP_REQUEST1;

				// -----------------------------------------------------------------------------------------------------------
				// Save image from camera
			ELSIF gVisionImage.CMD.SaveImage THEN
				// Generate file name if not provided
				IF gVisionImage.CFG.FileName = '' THEN
					// Generate new file name
					DTGetTime_0.enable := 1;
					DTGetTime_0();
					DT_TO_DTStructure(DTGetTime_0.DT1, ADR(DTStructure_0));
					FileNamePict := gVisionImage.CFG.DirName;
					brsstrcat(ADR(FileNamePict), ADR('/'));
					tmpStr := UINT_TO_STRING(DTStructure_0.year);
					brsstrcat(ADR(FileNamePict), ADR(tmpStr));
					brsstrcat(ADR(FileNamePict), ADR('_'));
					tmpStr := USINT_TO_STRING(DTStructure_0.month);
					IF(DTStructure_0.month < 10) THEN
						brsstrcat(ADR(FileNamePict), ADR('0'));
					END_IF
					brsstrcat(ADR(FileNamePict), ADR(tmpStr));
					brsstrcat(ADR(FileNamePict), ADR('_'));
					tmpStr := USINT_TO_STRING(DTStructure_0.day);
					IF(DTStructure_0.day < 10) THEN
						brsstrcat(ADR(FileNamePict), ADR('0'));
					END_IF
					brsstrcat(ADR(FileNamePict), ADR(tmpStr));
					brsstrcat(ADR(FileNamePict), ADR('_'));
					tmpStr := USINT_TO_STRING(DTStructure_0.hour);
					IF(DTStructure_0.hour < 10) THEN
						brsstrcat(ADR(FileNamePict), ADR('0'));
					END_IF
					brsstrcat(ADR(FileNamePict), ADR(tmpStr));
					brsstrcat(ADR(FileNamePict), ADR('_'));
					tmpStr := USINT_TO_STRING(DTStructure_0.minute);
					IF(DTStructure_0.minute < 10) THEN
						brsstrcat(ADR(FileNamePict), ADR('0'));
					END_IF
					brsstrcat(ADR(FileNamePict), ADR(tmpStr));
					brsstrcat(ADR(FileNamePict), ADR('_'));
					tmpStr := USINT_TO_STRING(DTStructure_0.second);
					IF(DTStructure_0.second < 10) THEN
						brsstrcat(ADR(FileNamePict), ADR('0'));
					END_IF
					brsstrcat(ADR(FileNamePict), ADR(tmpStr));
				ELSE
					FileNamePict := gVisionImage.CFG.FileName;
				END_IF

				brsstrcpy(ADR(FileNameSvg), ADR(FileNamePict));
				brsstrcat(ADR(FileNameSvg), ADR('.svg'));
				IF gVisionImage.CFG.ImageType = viBASE_IMAGE_TYPE_JPG THEN
					brsstrcat(ADR(FileNamePict), ADR('.jpg'));
				ELSE
					brsstrcat(ADR(FileNamePict), ADR('.bmp'));
				END_IF

				// Reset all function blocks
				FileCreate_0.enable := FALSE;
				FileCreate_0();
				FileWrite_0.enable := FALSE;
				FileWrite_0();
				FileClose_0.enable := FALSE;
				FileClose_0();
				ViBaseGetImage_0.Execute := FALSE;
				ViBaseGetImage_0();
				httpEncodeBase64_0.enable := FALSE;
				httpEncodeBase64_0();

				gVisionImage.DAT.Status		:= 65535;
				Step						:= VISTEP_REQUEST1;

			// -----------------------------------------------------------------------------------------------------------
			// Reset error
			ELSIF gVisionImage.CMD.ResetError THEN
				gVisionImage.CMD.ResetError := FALSE;
			END_IF

			// -----------------------------------------------------------------------------------------------------------
			// Load new image into window
			IF visImageSelectedOld <> gVisionImage.DAT.ImageSelected AND dir_entry > 0 THEN
				brsmemset(ADR(gVisionImage.DAT.ImagePath), 0, SIZEOF(gVisionImage.DAT.ImagePath));
				brsmemset(ADR(tmpStr), 0, SIZEOF(tmpStr));
				gVisionImage.DAT.ImagePath := '/FileDevice:';
				brsstrcat(ADR(gVisionImage.DAT.ImagePath), ADR(gVisionImage.CFG.FileDevice));
				brsstrcat(ADR(gVisionImage.DAT.ImagePath), ADR('/'));
				brsstrcat(ADR(gVisionImage.DAT.ImagePath), ADR(gVisionImage.CFG.DirName));
				brsstrcat(ADR(gVisionImage.DAT.ImagePath), ADR('/'));
				brsstrcat(ADR(gVisionImage.DAT.ImagePath), ADR(gVisionImage.DAT.ImageSelected));
			END_IF
			IF dir_entry = 0 THEN
				brsmemset(ADR(gVisionImage.DAT.ImagePath), 0, SIZEOF(gVisionImage.DAT.ImagePath));
			END_IF
			visImageSelectedOld := gVisionImage.DAT.ImageSelected;

		// -----------------------------------------------------------------------------------------------------------
		// Create directory on User-Partition, if not exists
		// -----------------------------------------------------------------------------------------------------------
		VISTEP_CREATE_DIR:
			DirCreate_0.enable	:= TRUE;
			DirCreate_0.pDevice	:= ADR(gVisionImage.CFG.FileDevice);
			DirCreate_0.pName	:= ADR(gVisionImage.CFG.DirName);
			DirCreate_0();

			IF DirCreate_0.status = 0 OR DirCreate_0.status = fiERR_DIR_ALREADY_EXIST THEN
				Step := VISTEP_READ_DIR1;
			ELSIF DirCreate_0.status <> 65535 THEN
				gVisionImage.DAT.Status := DirCreate_0.status;
				Step := VISTEP_ERR;
			END_IF

		// -----------------------------------------------------------------------------------------------------------
		// Delete directory on User-Partition
		// -----------------------------------------------------------------------------------------------------------
		VISTEP_DELETE_DIR:
			DirDeleteEx_0.enable	:= TRUE;
			DirDeleteEx_0.pDevice	:= ADR(gVisionImage.CFG.FileDevice);
			DirDeleteEx_0.pName		:= ADR(gVisionImage.CFG.DirName);
			DirDeleteEx_0();

			IF DirDeleteEx_0.status = 0 THEN
				Step := VISTEP_CREATE_DIR;
			ELSIF DirDeleteEx_0.status <> 65535 THEN
				gVisionImage.DAT.Status := DirDeleteEx_0.status;
				Step := VISTEP_ERR;
			END_IF

		// -----------------------------------------------------------------------------------------------------------
		// Read all existing image names from directory
		// -----------------------------------------------------------------------------------------------------------
		VISTEP_READ_DIR1:
			// Clear all memory
			brsmemset(ADR(gVisionImage.DAT.ImagesList), 0, SIZEOF(gVisionImage.DAT.ImagesList));
			brsmemset(ADR(gVisionImage.DAT.ImageSelected), 0, SIZEOF(gVisionImage.DAT.ImageSelected));
			visImageSelectedOld := '';
			gVisionImage.DAT.ImageSelected	:= '';
			dir_entry			:= 0;
			idx					:= 0;
			file_newest			:= '';
			file_oldest			:= '';
			date_newest			:= UDINT_TO_DT(0);
			date_oldest			:= DT#2100-06-06-12:00:00;
			cmdDeleteOldest		:= FALSE;
			Step := VISTEP_READ_DIR2;

		// -----------------------------------------------------------------------------------------------------------
		// Proceed with next entry
		// -----------------------------------------------------------------------------------------------------------
		VISTEP_READ_DIR2:
			DirRead_0.enable 	:= 1;
			DirRead_0.pDevice 	:= ADR(gVisionImage.CFG.FileDevice);
			DirRead_0.pPath		:= ADR(gVisionImage.CFG.DirName);
			DirRead_0.entry 	:= idx;
			DirRead_0.option 	:= fiFILE;
			DirRead_0.pData 	:= ADR(dir_data);
			DirRead_0.data_len 	:= SIZEOF(dir_data);
			DirRead_0();

			IF DirRead_0.status = 0 THEN
				// Make sure file is an image and we have space to store them
				IF  brsstrcmp(ADR(dir_data.Filename) + brsstrlen(ADR(dir_data.Filename)) - 4, ADR('.bmp')) = 0 OR
					brsstrcmp(ADR(dir_data.Filename) + brsstrlen(ADR(dir_data.Filename)) - 4, ADR('.jpg')) = 0 OR
					brsstrcmp(ADR(dir_data.Filename) + brsstrlen(ADR(dir_data.Filename)) - 4, ADR('.svg')) = 0 THEN
					// Find newest and oldest file
					IF dir_data.Date > date_newest THEN
						brsstrcpy(ADR(file_newest), ADR(dir_data.Filename));
						date_newest := dir_data.Date;
					END_IF
					IF dir_data.Date < date_oldest THEN
						brsstrcpy(ADR(file_oldest), ADR(dir_data.Filename));
						date_oldest := dir_data.Date;
					END_IF
					IF dir_entry <= SIZEOF(gVisionImage.DAT.ImagesList)/SIZEOF(gVisionImage.DAT.ImagesList[0]) - 1 THEN
						// Create list box data
						gVisionImage.DAT.ImagesList[dir_entry] := '{"value":"';
						brsstrcat(ADR(gVisionImage.DAT.ImagesList[dir_entry]), ADR(dir_data.Filename));
						brsstrcat(ADR(gVisionImage.DAT.ImagesList[dir_entry]), ADR('","text":"'));
						brsstrcat(ADR(gVisionImage.DAT.ImagesList[dir_entry]), ADR(dir_data.Filename));
						brsstrcat(ADR(gVisionImage.DAT.ImagesList[dir_entry]), ADR('"}'));
						dir_entry := dir_entry + 1;
					ELSE
						cmdDeleteOldest := TRUE;
					END_IF
				END_IF
				idx := idx + 1;
			ELSIF DirRead_0.status = fiERR_NO_MORE_ENTRIES THEN
				IF cmdDeleteOldest THEN
					brsstrcpy(ADR(tmpStr), ADR(gVisionImage.CFG.DirName));
					brsstrcat(ADR(tmpStr), ADR('/'));
					brsstrcat(ADR(tmpStr), ADR(file_oldest));
					Step := VISTEP_DELETE_IMAGE;
				ELSE
					TON_VisPause(IN := FALSE);
					Step := VISTEP_READ_DIR3;
				END_IF
			ELSIF DirRead_0.status <> 65535 THEN
				gVisionImage.DAT.Status := DirRead_0.status;
				Step := VISTEP_ERR;
			END_IF

		// -----------------------------------------------------------------------------------------------------------
		// Wait for vis before setting last file
		// -----------------------------------------------------------------------------------------------------------
		VISTEP_READ_DIR3:
			TON_VisPause.IN := TRUE;
			TON_VisPause.PT := T#250ms;
			TON_VisPause();

			IF TON_VisPause.Q THEN
				brsstrcpy(ADR(gVisionImage.DAT.ImageSelected), ADR(file_newest));
				brsmemset(ADR(gVisionImage.CMD), 0, SIZEOF(gVisionImage.CMD));
				Step := VISTEP_WAIT;
			END_IF

		// -----------------------------------------------------------------------------------------------------------
		// Delete Image
		// -----------------------------------------------------------------------------------------------------------
		VISTEP_DELETE_IMAGE:
			cmdDeleteOldest			:= FALSE;
			FileDelete_0.enable 	:= 1;
			FileDelete_0.pDevice	:= ADR(gVisionImage.CFG.FileDevice);
			FileDelete_0.pName 		:= ADR(FileNamePict);
			FileDelete_0();

			IF FileDelete_0.status = 0 THEN
				Step := VISTEP_READ_DIR1;
			ELSIF FileDelete_0.status <> 65535 THEN
				gVisionImage.DAT.Status := FileDelete_0.status;
				Step := VISTEP_ERR;
			END_IF

		// -----------------------------------------------------------------------------------------------------------
		// Get new image
		// -----------------------------------------------------------------------------------------------------------
		VISTEP_REQUEST1:
			ViBaseGetImage_0.MpLink := ADR(gVisionImage.CFG.ComponentLink);
			ViBaseGetImage_0.Execute := TRUE;
			IF gVisionImage.CMD.GetImage THEN
				ViBaseGetImage_0.Type :=  viBASE_IMAGE_TYPE_JPG;
				ViBaseGetImage_0.QualityLevel := IMAGE_QUALITY;
			ELSE
				ViBaseGetImage_0.Type :=  gVisionImage.CFG.ImageType;
				ViBaseGetImage_0.QualityLevel := gVisionImage.CFG.ImageQuality;
			END_IF
			ViBaseGetImage_0.Timeout := T#10s;
			ViBaseGetImage_0.Buffer := ADR(bufferImage);
			ViBaseGetImage_0.BufferSize := SIZEOF(bufferImage);;
			ViBaseGetImage_0();

			IF ViBaseGetImage_0.Busy = 0 THEN
				IF ViBaseGetImage_0.StatusID = 0 THEN
					Step := VISTEP_REQUEST2;
				ELSIF ViBaseGetImage_0.StatusID <> ERR_FUB_BUSY THEN
					gVisionImage.DAT.Status := ViBaseGetImage_0.StatusID;
					Step := VISTEP_ERR;
				END_IF
			END_IF

		// -----------------------------------------------------------------------------------------------------------
		// Convert to base64
		// -----------------------------------------------------------------------------------------------------------
		VISTEP_REQUEST2:
			httpEncodeBase64_0.enable    := TRUE;
			httpEncodeBase64_0.pSrc      := ADR(bufferImage);
			httpEncodeBase64_0.srcLen    := ViBaseGetImage_0.BufferLen;
			httpEncodeBase64_0.pDest     := ADR(bufferImage64);
			httpEncodeBase64_0.destSize  := SIZEOF(bufferImage64);
			httpEncodeBase64_0();

			IF httpEncodeBase64_0.status = 0 THEN
				Step := VISTEP_REQUEST3;
			ELSIF httpEncodeBase64_0.status <> ERR_FUB_BUSY THEN
				gVisionImage.DAT.Status := httpEncodeBase64_0.status;
				Step := VISTEP_ERR;
			END_IF

		// -----------------------------------------------------------------------------------------------------------
		// Create SVG data
		// -----------------------------------------------------------------------------------------------------------
		VISTEP_REQUEST3:
			brsmemset(ADR(visCameraImage), 0, SIZEOF(visCameraImage));
			visCameraImage := '<svg xmlns="http://www.w3.org/2000/svg" xml:space="preserve" width="';
			brsitoa(IMAGE_WIDTH, ADR(tmpStr));
			brsstrcat(ADR(visCameraImage), ADR(tmpStr));
			brsstrcat(ADR(visCameraImage), ADR('px" height="'));
			brsitoa(IMAGE_HEIGHT, ADR(tmpStr));
			brsstrcat(ADR(visCameraImage), ADR(tmpStr));
			brsstrcat(ADR(visCameraImage), ADR('px" shape-rendering="geometricPrecision" text-rendering="geometricPrecision" image-rendering="optimizeQuality" fill-rule="nonzero" clip-rule="evenodd" viewBox="0 0 '));
			brsitoa(gVisionImage.CFG.ImageWidth, ADR(tmpStr));
			brsstrcat(ADR(visCameraImage), ADR(tmpStr));
			brsstrcat(ADR(visCameraImage), ADR(' '));
			brsitoa(gVisionImage.CFG.ImageHeight, ADR(tmpStr));
			brsstrcat(ADR(visCameraImage), ADR(tmpStr));
			brsstrcat(ADR(visCameraImage), ADR('" xmlns:xlink="http://www.w3.org/1999/xlink"><image xlink:href="data:image/'));
			IF ViBaseGetImage_0.Type = viBASE_IMAGE_TYPE_JPG THEN
				brsstrcat(ADR(visCameraImage), ADR('jpeg'));
			ELSIF ViBaseGetImage_0.Type = viBASE_IMAGE_TYPE_BMP THEN
				brsstrcat(ADR(visCameraImage), ADR('bmp'));
			END_IF
			brsstrcat(ADR(visCameraImage), ADR(';base64,'));
			brsstrcat(ADR(visCameraImage), ADR(bufferImage64));
			brsstrcat(ADR(visCameraImage), ADR('"/>'));

			// Finish up when command was get image
			IF gVisionImage.CMD.GetImage THEN
				brsstrcat(ADR(visCameraImage), ADR('</svg>'));
				gVisionImage.CMD.GetImage := FALSE;
				Step := VISTEP_WAIT;
			// Save image to PLC
			ELSE
				bufferAdr := ADR(bufferImage);
				bufferLen := ViBaseGetImage_0.BufferLen;
				Step := VISTEP_SAVE1;
			END_IF

		// -----------------------------------------------------------------------------------------------------------
		// Save image
		// -----------------------------------------------------------------------------------------------------------
		VISTEP_SAVE1:
			FileCreate_0.enable		:= TRUE;
			FileCreate_0.pDevice	:= ADR(gVisionImage.CFG.FileDevice);
			FileCreate_0.pFile		:= ADR(FileNamePict);
			FileCreate_0();

			IF FileCreate_0.status = 0 THEN
				Step := VISTEP_SAVE2;
			ELSIF FileCreate_0.status <> ERR_FUB_BUSY THEN
				gVisionImage.DAT.Status := FileCreate_0.status;
				Step := VISTEP_ERR;
			END_IF

		VISTEP_SAVE2:
			FileWrite_0.enable		:= TRUE;
			FileWrite_0.ident		:= FileCreate_0.ident;
			FileWrite_0.pSrc		:= bufferAdr;
			FileWrite_0.len			:= bufferLen;
			FileWrite_0();

			IF FileWrite_0.status = 0 THEN
				Step := VISTEP_SAVE3;
			ELSIF FileWrite_0.status <> ERR_FUB_BUSY THEN
				gVisionImage.DAT.Status := FileWrite_0.status;
				Step := VISTEP_ERR;
			END_IF

		VISTEP_SAVE3:
			FileClose_0.enable		:= TRUE;
			FileClose_0.ident		:= FileCreate_0.ident;
			FileClose_0();

			IF FileClose_0.status = 0 THEN
				IF bufferAdr = ADR(bufferImage) THEN
					Step := VISTEP_SVG_CROSSH;
				ELSE
					Step := VISTEP_READ_DIR1;
				END_IF
			ELSIF FileClose_0.status <> ERR_FUB_BUSY THEN
				gVisionImage.DAT.Status := FileClose_0.status;
				Step := VISTEP_ERR;
			END_IF

		// -----------------------------------------------------------------------------------------------------------
		// Prepare the second part after base64 picture data
		VISTEP_SVG_CROSSH:
			brsmemset(ADR(bufferCrosshair), 0, SIZEOF(bufferCrosshair));
			brsstrcat(ADR(bufferCrosshair), ADR('<defs><symbol id="Fadenkreuz"><desc>Ein einfaches Fadenkreuz</desc><g id="Crosshair"><path style="stroke:#ff0000;stroke-width:5" d="M 40,1 V 30 Z" id="up" /><path style="stroke:#ff0000;stroke-width:5" d="M 40,50 V 80 Z" id="down" /><path style="stroke:#ff0000;stroke-width:5" d="M 30,40 H 0 Z" id="left" /><path style="stroke:#ff0000;stroke-width:5" d="M 80,40 H 50 Z" id="right" /><circle style="fill:none;stroke:#ff0000;stroke-width:5" cx="40" cy="40" r="25" id="circle6" /></g></symbol></defs>'));

			FOR idx := 1 TO MAX_NUM_RESULTS DO
				IF (gVisionImage.DAT.Crosshair[idx].CrosshairX <> 0 AND gVisionImage.DAT.Crosshair[idx].CrosshairY <> 0) AND (brsstrlen(ADR(bufferCrosshair)) < SIZEOF(bufferCrosshair) - 100) THEN
					brsstrcat(ADR(bufferCrosshair), ADR('<use xlink:href="#Fadenkreuz" transform="translate('));
					brsitoa(REAL_TO_DINT(gVisionImage.DAT.Crosshair[idx].CrosshairX), ADR(tmpStr));
					brsstrcat(ADR(bufferCrosshair), ADR(tmpStr));
					brsstrcat(ADR(bufferCrosshair), ADR(','));
					brsitoa(REAL_TO_DINT(gVisionImage.DAT.Crosshair[idx].CrosshairY), ADR(tmpStr));
					brsstrcat(ADR(bufferCrosshair), ADR(tmpStr));
					brsstrcat(ADR(bufferCrosshair), ADR(') rotate('));
					brsitoa(REAL_TO_DINT(gVisionImage.DAT.Crosshair[idx].CrosshairRotate), ADR(tmpStr));
					brsstrcat(ADR(bufferCrosshair), ADR(tmpStr));
					brsstrcat(ADR(bufferCrosshair), ADR(',40,40)"/>'));
				END_IF
			END_FOR
			Step := VISTEP_SVG_CONCAT;

		VISTEP_SVG_CONCAT:
			// Reset all function blocks
			FileCreate_0.enable := FALSE;
			FileCreate_0();
			FileWrite_0.enable := FALSE;
			FileWrite_0();
			FileClose_0.enable := FALSE;
			FileClose_0();

			brsstrcat(ADR(visCameraImage), ADR(bufferCrosshair));
			brsstrcat(ADR(visCameraImage), ADR('</svg>'));
			bufferAdr := ADR(visCameraImage);
			bufferLen := brsstrlen(ADR(visCameraImage));
			FileNamePict := FileNameSvg;

			Step := VISTEP_SAVE1;

			// -----------------------------------------------------------------------------------------------------------
			// Error state
			// -----------------------------------------------------------------------------------------------------------
		VISTEP_ERR:
			// Reset all function blocks
			FileCreate_0.enable := FALSE;
			FileCreate_0();
			FileWrite_0.enable := FALSE;
			FileWrite_0();
			FileClose_0.enable := FALSE;
			FileClose_0();
			FileDelete_0.enable := FALSE;
			FileDelete_0();

			ViBaseGetImage_0.Execute := FALSE;
			ViBaseGetImage_0();
			httpEncodeBase64_0.enable := FALSE;
			httpEncodeBase64_0();

			IF gVisionImage.CMD.ResetError THEN
				gVisionImage.CMD.ResetError := FALSE;
				Step := VISTEP_WAIT;
			END_IF
			brsmemset(ADR(gVisionImage.CMD), 0, SIZEOF(gVisionImage.CMD));
	END_CASE

END_PROGRAM
```

### Program Logical/Vision/Vi_visu

#### Variables.var
```iecst
(*-----------------------------------------------------------------------------------------------------------------------------------------*)
(*Main vision and data structures*)
VAR
	VisionSensor : REFERENCE TO typVisionMain; (*General vision functions that are independent from the inspection function*)
	VisionLight : REFERENCE TO typLightMain; (*General vision functions that are independent from the inspection function*)
	Match : REFERENCE TO typMatchMain; (*Data that is specific for the match function*)
	CodeReader : REFERENCE TO typCodeReaderMain; (*Data that is specific for the code reader*)
	MT : REFERENCE TO typMTMain; (*Data that is specific for the MT function*)
	OCR : REFERENCE TO typOCRMain; (*Data that is specific for the OCR function*)
	DOCR : REFERENCE TO typDOCRMain; (*Data that is specific for the OCR function*)
	Blob : REFERENCE TO typBlobMain; (*Data that is specific for the blob function*)
	Pixel : REFERENCE TO typPixelMain; (*Data that is specific for the blob function*)
	tmpMatch : {REDUND_UNREPLICABLE} typMatchMain; (*Data that is specific for the match function*)
	tmpCodeReader : {REDUND_UNREPLICABLE} typCodeReaderMain; (*Data that is specific for the code reader*)
	tmpMT : {REDUND_UNREPLICABLE} typMTMain; (*Data that is specific for the OCR function*)
	tmpOCR : {REDUND_UNREPLICABLE} typOCRMain; (*Data that is specific for the OCR function*)
	tmpDOCR : {REDUND_UNREPLICABLE} typDOCRMain; (*Data that is specific for the OCR function*)
	tmpBlob : {REDUND_UNREPLICABLE} typBlobMain; (*Data that is specific for the blob function*)
	tmpPixel : {REDUND_UNREPLICABLE} typPixelMain; (*Data that is specific for the blob function*)
END_VAR
(*-----------------------------------------------------------------------------------------------------------------------------------------*)
(*Sensor variables*)
VAR
	visSensorEnableCommand : BOOL; (*Enable/Disable vision trigger and enable when camera is not ready*)
	visEnableSetup : BOOL; (*Enable/Disable vision setup when camera is not ready*)
	visEnableRepetitive : BOOL; (*Enable/Disable repetitive mode*)
	visImageTrigger : BOOL; (*Trigger new image*)
	visSensorFlashColor : STRING[10]; (*Flash color string*)
	visSensorFlashColorOld : STRING[10]; (*Flash color string*)
	visSelectedFlashSegment : ARRAY[0..3] OF USINT := [4(1)]; (*Selected flash segments*)
	visSelectedFlashSegmentOld : ARRAY[0..3] OF USINT := [4(1)]; (*Selected flash segments*)
	visRepetitiveMode : BOOL; (*Enable/Disable repetitive mode*)
	RepetitiveModeTimer : TON; (*Timer for repetitive mode*)
	InitialSearchSensor : BOOL; (*Flag for first boot*)
	AutoSetupRunning : ARRAY[1..MAX_NUM_CAMS] OF BOOL; (*Flag for auto setup running*)
END_VAR
(*-----------------------------------------------------------------------------------------------------------------------------------------*)
(*Lights variables*)
VAR
	InitialSearchLight : BOOL;
	visLightsTrigger : BOOL;
	visLightsReset : BOOL;
	visLightsEnableCommand : BOOL;
	visLightsFlashColor : STRING[10]; (*Flash color string*)
	visLightsFlashColorOld : STRING[10];
	visEnableLightBarValues : BOOL;
END_VAR
(*-----------------------------------------------------------------------------------------------------------------------------------------*)
(*Code Reader*)
VAR
	visSelectedCodeTypeDetected : ARRAY[1..MAX_NUM_RESULTS] OF STRING[80]; (*HMI helper string*)
	visSelectedCodeType : STRING[80]; (*HMI helper string*)
	visSelectedCodeTypeOld : STRING[80]; (*HMI helper string*)
	visSelectedParameterMode : STRING[80]; (*HMI helper string*)
	visSelectedParameterModeOld : STRING[80]; (*HMI helper string*)
	visCodeTypePresentDropDownValues : ARRAY[0..MAX_NUM_CODETYPES] OF STRING[80];
END_VAR
(*-----------------------------------------------------------------------------------------------------------------------------------------*)
(*Image, crosshair data and constants*)
VAR
	visCrossHair : typCrossHair; (*Data structure to draw the crosshairs on the main page*)
	CrosshairModelNumber : USINT;
	CrosshairPositionX : REAL;
	CrosshairPositionY : REAL;
	CrosshairOrientation : INT;
	tmpStr1 : STRING[1000];
	tmpStr2 : STRING[100];
	tmpStr3 : STRING[100];
	tmpC : REAL;
	tmpYI : REAL;
	tmpXI : REAL;
	DetailsNoOld : USINT;
	visTableNo : ARRAY[1..MAX_NUM_RESULTS] OF USINT := [1,2,3,4,5,6,7,8,9,10];
	i : UINT;
	visCameraStatus : STRING[30];
END_VAR
```

#### Main.st
```iecst
// --------------------------------------------------------------------------------------------------------------------
// This is a support task for the mappView visualization. The following functions are implemneted
// - Disable mappView functions when camera is not ready, available
// - Transfer parameters after vision setup
// Version 2.x (Check revision history for details)
// --------------------------------------------------------------------------------------------------------------------
PROGRAM _INIT
	// -----------------------------------------------------------------------------------------------------------
	// Map global structure to local reference
	VisionSensor ACCESS ADR(gVisionSensor[gSelectedSensor]);
	Blob ACCESS ADR(tmpBlob);
	CodeReader ACCESS ADR(tmpCodeReader);
	Match ACCESS ADR(tmpMatch);
	MT ACCESS ADR(tmpMT);
	OCR ACCESS ADR(tmpOCR);
	DOCR ACCESS ADR(tmpDOCR);
	Pixel ACCESS ADR(tmpPixel);

	// Map global structure to local reference
	VisionLight ACCESS ADR(gVisionLight[gSelectedLight]);

	// -----------------------------------------------------------------------------------------------------------
	// Preload code types
	FOR i := 0 TO MAX_NUM_CODETYPES DO
		IF CodeTypes[i] <> '' THEN
			brsstrcat(ADR(visCodeTypePresentDropDownValues[i]), ADR('{"value":"'));
			brsitoa(i, ADR(tmpStr1));
			brsstrcat(ADR(visCodeTypePresentDropDownValues[i]), ADR(tmpStr1));
			brsstrcat(ADR(visCodeTypePresentDropDownValues[i]), ADR('","text":"'));
			brsstrcat(ADR(visCodeTypePresentDropDownValues[i]), ADR(CodeTypes[i]));
			brsstrcat(ADR(visCodeTypePresentDropDownValues[i]), ADR('"}'));
		END_IF
	END_FOR

	// -----------------------------------------------------------------------------------------------------------
	visTableNo;
	InitialSearchSensor := TRUE;
	InitialSearchLight := TRUE;
	brsmemset(ADR(visCrossHair.SvgContent), 0, SIZEOF(visCrossHair.SvgContent));
	brsmemset(ADR(visCrossHair.SvgTransformation), 0, SIZEOF(visCrossHair.SvgTransformation));
	brsmemset(ADR(visCrossHair.SvgVisible), 0, SIZEOF(visCrossHair.SvgVisible));

END_PROGRAM

// -----------------------------------------------------------------------------------------------------------
// Cyclic part
// -----------------------------------------------------------------------------------------------------------
PROGRAM _CYCLIC
	// Select first available camera after reboot
	IF InitialSearchSensor THEN
		FOR i := 1 TO MAX_NUM_CAMS DO
			IF gVisionSensor[i].HW.Connected THEN
				gSelectedSensor := i;
				InitialSearchSensor := FALSE;
				EXIT;
			END_IF
		END_FOR
	END_IF

	// -----------------------------------------------------------------------------------------------------------
	// Map global structure to local reference for mappView
	// -----------------------------------------------------------------------------------------------------------
	// Make sure we dont exceed array limit
	IF(gSelectedSensor > MAX_NUM_CAMS) THEN
		gSelectedSensor := 1;
	END_IF
	IF(gSelectedSensor < 1) THEN
		gSelectedSensor := MAX_NUM_CAMS;
	END_IF

	// Assign pointers
	VisionSensor ACCESS ADR(gVisionSensor[gSelectedSensor]);
	IF(VisionSensor.CFG.DataStructure <> 0) THEN
		CASE VisionSensor.CFG.VisionFunction OF
			enumBlob:			Blob ACCESS VisionSensor.CFG.DataStructure;
			enumCoderReader:	CodeReader ACCESS VisionSensor.CFG.DataStructure;
			enumMatch:			Match ACCESS VisionSensor.CFG.DataStructure;
			enumMeasurement:	MT ACCESS VisionSensor.CFG.DataStructure;
			enumOCR:			OCR ACCESS VisionSensor.CFG.DataStructure;
			enumDOCR:			DOCR ACCESS VisionSensor.CFG.DataStructure;
			enumPixelCounter:	Pixel ACCESS VisionSensor.CFG.DataStructure;
		END_CASE
	ELSE
		RETURN;
	END_IF

	// Display camera status
	visCameraStatus := VisionSensor.DAT.StatusText;

	// -----------------------------------------------------------------------------------------------------------
	// Code Reader - selected/detected types
	// -----------------------------------------------------------------------------------------------------------
	IF VisionSensor.CFG.VisionFunction = enumCoderReader THEN
		IF visSelectedCodeType <> visSelectedCodeTypeOld THEN
			CodeReader.CodeType := UDINT_TO_USINT(brsatoi(ADR(visSelectedCodeType)));
		ELSE
			brsitoa(CodeReader.CodeType, ADR(visSelectedCodeType));
		END_IF
		visSelectedCodeTypeOld := visSelectedCodeType;
		IF visSelectedParameterMode <> visSelectedParameterModeOld THEN
			CodeReader.ParameterMode := UDINT_TO_USINT(brsatoi(ADR(visSelectedParameterMode)));
		ELSE
			brsitoa(CodeReader.ParameterMode, ADR(visSelectedParameterMode));
		END_IF
		visSelectedParameterModeOld := visSelectedParameterMode;
		FOR i := 1 TO MAX_NUM_RESULTS DO
			IF CodeReader.BarcodeType[i] <> 0 THEN
				brsstrcpy(ADR(visSelectedCodeTypeDetected[i]), ADR(CodeTypes[LIMIT(0, CodeReader.BarcodeType[i], MAX_NUM_CODETYPES)]));
			ELSE
				brsstrcpy(ADR(visSelectedCodeTypeDetected[i]), ADR(''));
			END_IF
		END_FOR
	END_IF

	// -----------------------------------------------------------------------------------------------------------
	// Translate flash color and segments from mappView to IO mapping
	// -----------------------------------------------------------------------------------------------------------
	IF visSensorFlashColor <> visSensorFlashColorOld THEN
		VisionSensor.DAT.FlashColor := UDINT_TO_USINT(brsatoi(ADR(visSensorFlashColor)));
	ELSE
		brsitoa(VisionSensor.DAT.FlashColor, ADR(visSensorFlashColor));
	END_IF
	visSensorFlashColorOld := visSensorFlashColor;
	IF brsmemcmp(ADR(visSelectedFlashSegment), ADR(visSelectedFlashSegmentOld), SIZEOF(visSelectedFlashSegment)) <> 0 THEN // The flash segments was changed in the mappView visualization
		VisionSensor.DAT.FlashSegment := SHL(visSelectedFlashSegment[0], 0) OR SHL(visSelectedFlashSegment[1], 1) OR SHL(visSelectedFlashSegment[2], 2) OR SHL(visSelectedFlashSegment[3], 3);
	ELSE
		visSelectedFlashSegment[0] := VisionSensor.DAT.FlashSegment.0;
		visSelectedFlashSegment[1] := VisionSensor.DAT.FlashSegment.1;
		visSelectedFlashSegment[2] := VisionSensor.DAT.FlashSegment.2;
		visSelectedFlashSegment[3] := VisionSensor.DAT.FlashSegment.3;
	END_IF
	visSelectedFlashSegmentOld := visSelectedFlashSegment;

	// -----------------------------------------------------------------------------------------------------------
	// Disable command buttons when camera is disconnected, not ready, processing an image or vision cockpit is open
	// -----------------------------------------------------------------------------------------------------------
	IF(NOT VisionSensor.HW.Connected OR NOT VisionSensor.HW.Ready OR VisionSensor.DAT.ImageProcessingActive OR VisionSensor.DAT.CockpitIsActive) THEN
		visSensorEnableCommand := FALSE;
	ELSE
		visSensorEnableCommand := TRUE;
	END_IF

	// -----------------------------------------------------------------------------------------------------------
	// Disable setup buttons when camera is disconnected, processing an image or not ready
	// -----------------------------------------------------------------------------------------------------------
	IF(NOT VisionSensor.HW.Connected OR NOT (VisionSensor.HW.Ready OR AutoSetupRunning[gSelectedSensor]) OR VisionSensor.DAT.ImageProcessingActive) THEN
		visEnableSetup := FALSE;
	ELSE
		visEnableSetup := TRUE;
	END_IF

	// -----------------------------------------------------------------------------------------------------------
	// Fire trigger for camera image
	// -----------------------------------------------------------------------------------------------------------
	IF((visImageTrigger OR EDGEPOS(VisionSensor.DAT.Enable)) AND VisionSensor.HW.Ready AND NOT VisionSensor.DAT.ImageProcessingActive) THEN
		// Add default delay and fire trigger
		IF NETTIME_ENABLE THEN
			VisionSensor.DAT.NettimeDelay := NettimeCurrent_us + NETTIME_DEFAULT_DELAY;
		END_IF
		// Hide previous results
		FOR i := 1 TO MAX_NUM_RESULTS DO
			visCrossHair.SvgVisible[i] := FALSE;
		END_FOR;
		VisionSensor.CMD.ImageTrigger	:= TRUE;
		visImageTrigger					:= FALSE;
		VisionSensor.DAT.Active			:= TRUE;
	END_IF

	// -----------------------------------------------------------------------------------------------------------
	// Get image from camera
	// -----------------------------------------------------------------------------------------------------------
	IF EDGENEG(VisionSensor.CMD.ImageTrigger) THEN
		gVisionImage.CFG.ComponentLink := gVisionSensor[gSelectedSensor].CFG.ComponentLink;
		gVisionImage.CFG.ImageHeight := gVisionSensor[gSelectedSensor].CFG.ResolutionHeight;
		gVisionImage.CFG.ImageWidth := gVisionSensor[gSelectedSensor].CFG.ResolutionWidth;
		gVisionImage.CMD.GetImage := TRUE;
	END_IF

	// -----------------------------------------------------------------------------------------------------------
	// Repetitive mode
	// -----------------------------------------------------------------------------------------------------------
	visEnableRepetitive := visSensorEnableCommand OR visRepetitiveMode;
	IF visRepetitiveMode THEN
		RepetitiveModeTimer.IN := TRUE;
		IF RepetitiveModeTimer.Q THEN
			IF VisionSensor.HW.Ready AND NOT VisionSensor.DAT.ImageProcessingActive THEN
				IF NETTIME_ENABLE THEN
					VisionSensor.DAT.NettimeDelay := NettimeCurrent_us + NETTIME_DEFAULT_DELAY;
				END_IF
				RepetitiveModeTimer.IN := FALSE;
				VisionSensor.CMD.ImageTrigger := TRUE;
			END_IF
		END_IF
		VisionSensor.DAT.Enable := FALSE;
	ELSE
		RepetitiveModeTimer.IN := TRUE;
	END_IF
	RepetitiveModeTimer(PT := T#1000ms);

	// -----------------------------------------------------------------------------------------------------------
	// Select first available light after reboot
	// -----------------------------------------------------------------------------------------------------------
	IF InitialSearchLight THEN
		FOR i := 1 TO MAX_NUM_LIGHTS DO
			IF gVisionLight[i].HW.Connected THEN
				gSelectedLight := i;
				InitialSearchLight := FALSE;
				EXIT;
			END_IF
		END_FOR
	END_IF

	// -----------------------------------------------------------------------------------------------------------
	// Map global structure to local reference
	// -----------------------------------------------------------------------------------------------------------
	// Make sure we dont exceed array limit
	IF(gSelectedLight > MAX_NUM_LIGHTS) THEN
		gSelectedLight := 1;
	END_IF
	IF(gSelectedLight < 1) THEN
		gSelectedLight := MAX_NUM_LIGHTS;
	END_IF
	VisionLight ACCESS ADR(gVisionLight[gSelectedLight]);

	// -----------------------------------------------------------------------------------------------------------
	// Translate flash color from mappView to IO mapping
	// -----------------------------------------------------------------------------------------------------------
	// Hint: Normally copy from recipe (VisionLight) to visu. Only in case of a change in the visu copy to recipe
	IF visLightsFlashColor <> visLightsFlashColorOld THEN // The flash color was changed in the mappView visualization
		VisionLight.DAT.FlashColor := UDINT_TO_USINT(brsatoi(ADR(visLightsFlashColor)));
	ELSE
		brsitoa(VisionLight.DAT.FlashColor, ADR(visLightsFlashColor));
	END_IF
	visLightsFlashColorOld := visLightsFlashColor;

	// -----------------------------------------------------------------------------------------------------------
	// Reset Light trigger manually
	// -----------------------------------------------------------------------------------------------------------
	IF (visLightsReset) THEN
		VisionLight.CMD.FlashTrigger := FALSE;
		visLightsReset := FALSE;
	END_IF

	// -----------------------------------------------------------------------------------------------------------
	// Fire trigger for lights
	// -----------------------------------------------------------------------------------------------------------
	IF(visLightsTrigger AND VisionLight.HW.Ready) THEN
		// Add default delay and fire trigger
		IF NETTIME_ENABLE THEN
			VisionLight.DAT.NettimeDelay := NettimeCurrent_us + NETTIME_DEFAULT_DELAY;
		END_IF
		VisionLight.CMD.FlashTrigger := TRUE;
		visLightsTrigger := FALSE;
	END_IF

	// -----------------------------------------------------------------------------------------------------------
	// Disable command button when light is disconnected or not ready
	// -----------------------------------------------------------------------------------------------------------
	IF(NOT VisionLight.HW.Connected OR NOT VisionLight.HW.Ready) THEN
		visLightsEnableCommand := FALSE;
	ELSE
		visLightsEnableCommand := TRUE;
	END_IF

	// -----------------------------------------------------------------------------------------------------------
	// Enable fields for different light types
	// -----------------------------------------------------------------------------------------------------------
	visEnableLightBarValues := VisionLight.CFG.LightType = enumLightbar;

	// -----------------------------------------------------------------------------------------------------------
	// Draw cross hairs on main page
	// -----------------------------------------------------------------------------------------------------------
	IF (EDGENEG(gVisionImage.CMD.GetImage) AND visCrossHair.ShowCrosshair) OR EDGEPOS(visCrossHair.ShowCrosshair) OR (visCrossHair.DetailsNo <> DetailsNoOld) THEN
		// -----------------------------------------------------------------------------------------------------------
		// Handle details no
		IF(visCrossHair.DetailsNo < 1) THEN
			visCrossHair.DetailsNo := VisionSensor.DAT.ResultCnt;
		END_IF
		IF(visCrossHair.DetailsNo > VisionSensor.DAT.ResultCnt) THEN
			visCrossHair.DetailsNo := 1;
		END_IF
		IF visCrossHair.PixelRatio = 0 THEN
			visCrossHair.PixelRatio := 100;
		END_IF
		DetailsNoOld := visCrossHair.DetailsNo;
		brsmemset(ADR(gVisionImage.DAT.Crosshair), 0, SIZEOF(gVisionImage.DAT.Crosshair));

		// -----------------------------------------------------------------------------------------------------------
		// Create cross hairs and data for all results
		FOR i := 1 TO MAX_NUM_RESULTS DO
			visCrossHair.SvgTransformation[i] := '';
			visCrossHair.SvgVisible[i] := FALSE;
			CrosshairPositionX := 0;
			CrosshairPositionY := 0;
			gVisionImage.DAT.Crosshair[i].CrosshairX		:= 0;
			gVisionImage.DAT.Crosshair[i].CrosshairY		:= 0;
			gVisionImage.DAT.Crosshair[i].CrosshairRotate	:= 0;
			brsmemset(ADR(gVisionImage.DAT.Crosshair[i].Text), 0, SIZEOF(gVisionImage.DAT.Crosshair[i].Text));

			// -----------------------------------------------------------------------------------------------------------
			// Make sure we have data to display
			IF(VisionSensor.DAT.ResultCnt <> 0 AND i <= VisionSensor.DAT.ResultCnt) THEN
				// Select data source from vision function
				CASE VisionSensor.CFG.VisionFunction OF
					enumBlob:
						CrosshairModelNumber := gBlob.ModelNumber[i];
						CrosshairPositionX := UDINT_TO_REAL(gBlob.PositionX[i])/UINT_TO_REAL(gVisionSensor[gSelectedSensor].CFG.ResolutionWidth)*1280;
						CrosshairPositionY := UDINT_TO_REAL(gBlob.PositionY[i])/UINT_TO_REAL(gVisionSensor[gSelectedSensor].CFG.ResolutionHeight)*1024;
						CrosshairOrientation := gBlob.Orientation[i];
					enumMatch:
						CrosshairModelNumber := gMatch.ModelNumber[i];
						CrosshairPositionX := UDINT_TO_REAL(gMatch.PositionX[i])/UINT_TO_REAL(gVisionSensor[gSelectedSensor].CFG.ResolutionWidth)*1280;
						CrosshairPositionY := UDINT_TO_REAL(gMatch.PositionY[i])/UINT_TO_REAL(gVisionSensor[gSelectedSensor].CFG.ResolutionHeight)*1024;
						CrosshairOrientation := gMatch.Orientation[i];
					enumCoderReader:
						CrosshairPositionX := UDINT_TO_REAL(gCodeReader.PositionX[i])/UINT_TO_REAL(gVisionSensor[gSelectedSensor].CFG.ResolutionWidth)*1280;
						CrosshairPositionY := UDINT_TO_REAL(gCodeReader.PositionY[i])/UINT_TO_REAL(gVisionSensor[gSelectedSensor].CFG.ResolutionHeight)*1024;
						CrosshairOrientation := gCodeReader.Orientation[i];
					enumOCR:
						CrosshairPositionX := UDINT_TO_REAL(gOCR.PositionX[i])/UINT_TO_REAL(gVisionSensor[gSelectedSensor].CFG.ResolutionWidth)*1280;
						CrosshairPositionY := UDINT_TO_REAL(gOCR.PositionY[i])/UINT_TO_REAL(gVisionSensor[gSelectedSensor].CFG.ResolutionHeight)*1024;
						CrosshairOrientation := gOCR.Orientation[i];
					enumDOCR:
						CrosshairPositionX := UDINT_TO_REAL(gDOCR.PositionX[i])/UINT_TO_REAL(gVisionSensor[gSelectedSensor].CFG.ResolutionWidth)*1280;
						CrosshairPositionY := UDINT_TO_REAL(gDOCR.PositionY[i])/UINT_TO_REAL(gVisionSensor[gSelectedSensor].CFG.ResolutionHeight)*1024;
						CrosshairOrientation := gOCR.Orientation[i];
					enumMeasurement:
						IF(gMT.UseResultAsXY = TRUE) THEN
							CrosshairPositionX := UDINT_TO_REAL(gMT.Result[i])/10/UINT_TO_REAL(gVisionSensor[gSelectedSensor].CFG.ResolutionWidth)*1280;
							CrosshairPositionY := UDINT_TO_REAL(gMT.Result[i+1])/10/UINT_TO_REAL(gVisionSensor[gSelectedSensor].CFG.ResolutionHeight)*1024;
							i := i + 1;
						END_IF
				END_CASE

				// -----------------------------------------------------------------------------------------------------------
				// Show crosshair except for measurement function
				IF (VisionSensor.CFG.VisionFunction <> enumMeasurement OR gMT.UseResultAsXY = TRUE) THEN
					// -----------------------------------------------------------------------------------------------------------
					// Set start values
					IF(CrosshairPositionX <> 0 AND CrosshairPositionY <> 0) THEN
						visCrossHair.SvgVisible[i] := TRUE;

						// Highlight selected crosshair and show detailed information
						IF(visCrossHair.DetailsNo = i) THEN
							tmpStr1 := '[{"select":"#CrosshairBlue","display":false}, {"select":"#CrosshairRed","display":true, "translate":[';
						ELSE
							tmpStr1 := '[{"select":"#CrosshairRed","display":false}, { "select":"#CrosshairBlue","display":true, "translate":[';
						END_IF

						// Calculate cross hair X offset
						tmpXI := CrosshairPositionX / visCrossHair.PixelRatio;
						tmpC := USINT_TO_REAL(visCrossHair.Size) * visCrossHair.Scale / 2.0;
						brsitoa(REAL_TO_INT(tmpXI - tmpC), ADR(tmpStr2));
						brsstrcat(ADR(tmpStr1), ADR(tmpStr2));
						brsstrcat(ADR(tmpStr1), ADR(','));
						gVisionImage.DAT.Crosshair[i].CrosshairX := tmpXI - tmpC;

						// Calculate cross hair Y offset
						tmpYI := CrosshairPositionY / visCrossHair.PixelRatio;
						brsitoa(REAL_TO_INT(tmpYI - tmpC), ADR(tmpStr2));
						brsstrcat(ADR(tmpStr1), ADR(tmpStr2));
						gVisionImage.DAT.Crosshair[i].CrosshairY := tmpYI - tmpC;

						// Add cross hair scaling
						brsstrcat(ADR(tmpStr1), ADR('],"scale":['));
						brsftoa(visCrossHair.Scale, ADR(tmpStr2));
						brsstrcat(ADR(tmpStr1), ADR(tmpStr2));
						brsstrcat(ADR(tmpStr1), ADR(','));
						brsftoa(visCrossHair.Scale, ADR(tmpStr2));
						brsstrcat(ADR(tmpStr1), ADR(tmpStr2));

						// Add cross hair rotation
						brsstrcat(ADR(tmpStr1), ADR('],"spin":['));
						brsftoa(CrosshairOrientation/-100, ADR(tmpStr2));
						brsstrcat(ADR(tmpStr1), ADR(tmpStr2));
						brsstrcat(ADR(tmpStr1), ADR(','));
						brsitoa(visCrossHair.Size/2, ADR(tmpStr2));
						brsstrcat(ADR(tmpStr1), ADR(tmpStr2));
						brsstrcat(ADR(tmpStr1), ADR(','));
						brsstrcat(ADR(tmpStr1), ADR(tmpStr2));
						brsstrcat(ADR(tmpStr1), ADR(']}]'));
						visCrossHair.SvgTransformation[i] := tmpStr1;
						gVisionImage.DAT.Crosshair[i].CrosshairRotate := CrosshairOrientation/-100;

						// -----------------------------------------------------------------------------------------------------------
						// Add text data to selected cross hair
						IF(visCrossHair.DetailsNo = i) THEN
							tmpStr1 := '<text class="cText" fill="red" font-size="22" font-family="Helvetica, Arial, sans-serif" x="';
						ELSE
							tmpStr1 := '<text class="cText" fill="blue" font-size="22" font-family="Helvetica, Arial, sans-serif" x="';
						END_IF
						brsitoa(REAL_TO_INT(tmpXI - tmpC + visCrossHair.Size), ADR(tmpStr2));
						brsstrcat(ADR(tmpStr1), ADR(tmpStr2));
						brsstrcat(ADR(tmpStr1), ADR('" y="'));
						brsitoa(REAL_TO_INT(tmpYI - tmpC + visCrossHair.Size/2), ADR(tmpStr2));
						brsstrcat(ADR(tmpStr1), ADR(tmpStr2));
						brsstrcat(ADR(tmpStr1), ADR('"> '));

						// Create prototype for new entry
						tmpStr3:= '<tspan class="text" x="';
						brsitoa(REAL_TO_INT(tmpXI + tmpC), ADR(tmpStr2));
						brsstrcat(ADR(tmpStr3), ADR(tmpStr2));
						brsstrcat(ADR(tmpStr3), ADR('" dy="-5" >'));

						// Add result no information
						brsstrcat(ADR(tmpStr1), ADR(tmpStr3));
						brsitoa(i, ADR(tmpStr2));
						brsstrcat(ADR(tmpStr1), ADR(tmpStr2));
						brsstrcat(ADR(tmpStr1), ADR('</tspan></text>'));

						IF(visCrossHair.DetailsNo = i) THEN
							// -----------------------------------------------------------------------------------------------------------
							// Add text data from selected cross hair
							brsstrcat(ADR(tmpStr1), ADR('<text class="cText" fill="red" font-size="35" font-family="Helvetica, Arial, sans-serif" x="10" y="10"> '));

							// Add modell ID information for blob and match
							IF(VisionSensor.CFG.VisionFunction = enumBlob OR VisionSensor.CFG.VisionFunction = enumMatch) THEN
								CrosshairDetailsText(ADR(tmpStr1),  ADR('ID: '), CrosshairModelNumber);
							END_IF
							// Add X and Y position information
							IF(CrosshairPositionX <> 0) THEN
								CrosshairDetailsText(ADR(tmpStr1),  ADR('Pos X: '), CrosshairPositionX/visCrossHair.PixelRatio);
							END_IF
							IF(CrosshairPositionY <> 0) THEN
								CrosshairDetailsText(ADR(tmpStr1),  ADR('Pos Y: '), CrosshairPositionY/visCrossHair.PixelRatio);
							END_IF
							// Add orientation information
							IF(VisionSensor.CFG.VisionFunction <> enumMeasurement) THEN
								CrosshairDetailsText(ADR(tmpStr1),  ADR('Orientation: '), CrosshairOrientation/visCrossHair.PixelRatio);
							END_IF
							// Add detail information for blob
							IF(VisionSensor.CFG.VisionFunction = enumBlob AND gBlob.EnhancedBlobInformation = 1) THEN
								CrosshairDetailsText(ADR(tmpStr1),  ADR('Clipped: '), gBlob.Clipped[i]);
								CrosshairDetailsText(ADR(tmpStr1),  ADR('Gray: '), gBlob.MeanGrayValue[i]);
								CrosshairDetailsText(ADR(tmpStr1),  ADR('Length: '), UDINT_TO_REAL(gBlob.Length[i])/visCrossHair.PixelRatio);
								CrosshairDetailsText(ADR(tmpStr1),  ADR('Width: '), UDINT_TO_REAL(gBlob.Width[i])/visCrossHair.PixelRatio);
								CrosshairDetailsText(ADR(tmpStr1),  ADR('Area: '), UDINT_TO_REAL(gBlob.Area[i])/visCrossHair.PixelRatio);
							END_IF
							// Add detail information for match
							IF(VisionSensor.CFG.VisionFunction = enumMatch) THEN
								CrosshairDetailsText(ADR(tmpStr1),  ADR('Score: '), gMatch.Score[i]);
								CrosshairDetailsText(ADR(tmpStr1),  ADR('Scale: '), gMatch.Scale[i]);
							END_IF
							// Add detail information for code reader
							IF(VisionSensor.CFG.VisionFunction = enumCoderReader) THEN
								//CrosshairDetailsText(ADR(tmpStr1),  ADR('Code:'), UDINT_TO_REAL(CodeReader.BarcodeType[i]));
								tmpStr2:= '<tspan class="text" x="10" dy="32">';
								brsstrcat(ADR(tmpStr1), ADR(tmpStr2));
								brsstrcat(ADR(tmpStr1), ADR('Code: '));
								brsstrcat(ADR(tmpStr1), ADR(CodeTypes[LIMIT(0, gCodeReader.BarcodeType[i], MAX_NUM_CODETYPES)]));
								brsstrcat(ADR(tmpStr1), ADR('</tspan> '));
							END_IF
							brsstrcat(ADR(tmpStr1), ADR('</text>'));
						END_IF
					END_IF
					// -----------------------------------------------------------------------------------------------------------
					// Add result information measurement
				ELSE
					visCrossHair.SvgTransformation[i] := '[{"select":"#CrosshairRed","display":false}, {"select":"#CrosshairBlue","display":false}]';
					visCrossHair.SvgVisible[i] := TRUE;
					brsstrcpy(ADR(tmpStr1), ADR('<text class="cText" fill="red" font-size="35" font-family="Helvetica, Arial, sans-serif" x="10" y="'));
					brsitoa(i*40, ADR(tmpStr2));
					brsstrcat(ADR(tmpStr1), ADR(tmpStr2));
					brsstrcat(ADR(tmpStr1), ADR('"> '));
					CrosshairDetailsText(ADR(tmpStr1),  ADR('Result:'), UDINT_TO_REAL(gMT.Result[i])/1000);
					brsstrcat(ADR(tmpStr1), ADR('</text>'));
				END_IF
				visCrossHair.SvgContent[i] := tmpStr1;
				// for saving svg file
				brsstrcpy(ADR(gVisionImage.DAT.Crosshair[i].Text), ADR(tmpStr1));
			END_IF
		END_FOR
	END_IF
END_PROGRAM
```

### Program Logical/Vision/YourTask
